C01804=1030.164,-32.787,-88.307,167.818,43.138,158.004
C01805=1030.170,-32.537,-88.320,167.821,43.137,158.004
C01806=1030.176,-32.288,-88.333,167.824,43.135,158.004
C01807=1030.183,-32.038,-88.346,167.827,43.134,158.004
C01808=1030.190,-31.789,-88.359,167.829,43.132,158.004
C01809=1030.196,-31.539,-88.372,167.832,43.130,158.004
C01810=1030.202,-31.290,-88.385,167.834,43.129,158.004
C01811=1030.208,-31.040,-88.398,167.836,43.128,158.004
C01812=1030.214,-30.790,-88.411,167.839,43.126,158.004
C01813=1030.221,-30.540,-88.424,167.842,43.125,158.004
C01814=1030.227,-30.291,-88.438,167.845,43.123,158.004
C01815=1030.233,-30.042,-88.451,167.847,43.122,158.004
C01816=1030.239,-29.792,-88.464,167.850,43.120,158.004
C01817=1030.245,-29.543,-88.477,167.853,43.119,158.003
C01818=1030.252,-29.293,-88.490,167.856,43.117,158.003
C01819=1030.258,-29.044,-88.504,167.858,43.116,158.003
C01820=1030.264,-28.794,-88.516,167.860,43.114,158.003
C01821=1030.270,-28.544,-88.530,167.863,43.113,158.003
C01822=1030.277,-28.294,-88.544,167.866,43.111,158.003
C01823=1030.283,-28.045,-88.557,167.868,43.110,158.003
C01824=1030.289,-27.795,-88.570,167.871,43.108,158.003
C01825=1030.295,-27.546,-88.583,167.874,43.107,158.003
C01826=1030.302,-27.296,-88.596,167.877,43.105,158.003
C01827=1030.308,-27.046,-88.610,167.879,43.104,158.003
C01828=1030.314,-26.797,-88.623,167.881,43.102,158.003
C01829=1030.320,-26.548,-88.636,167.884,43.101,158.003
C01830=1030.326,-26.298,-88.651,167.887,43.099,158.002
C01831=1030.333,-26.048,-88.664,167.889,43.098,158.002
C01832=1030.339,-25.798,-88.676,167.892,43.097,158.002
C01833=1030.345,-25.549,-88.690,167.895,43.095,158.002
C01834=1030.351,-25.299,-88.704,167.897,43.094,158.002
C01835=1030.357,-25.050,-88.717,167.899,43.092,158.002
C01836=1030.363,-24.800,-88.730,167.902,43.091,158.002
C01837=1030.369,-24.551,-88.744,167.905,43.090,158.002
C01838=1030.376,-24.301,-88.758,167.908,43.088,158.002
C01839=1030.382,-24.052,-88.771,167.911,43.087,158.002
C01840=1030.388,-23.802,-88.784,167.912,43.085,158.002
C01841=1030.394,-23.552,-88.799,167.915,43.084,158.002
C01842=1030.400,-23.303,-88.812,167.918,43.083,158.002
C01843=1030.406,-23.054,-88.825,167.921,43.081,158.002
C01844=1030.413,-22.804,-88.838,167.923,43.080,158.002
C01845=1030.419,-22.554,-88.853,167.925,43.078,158.002
C01846=1030.425,-22.305,-88.866,167.928,43.077,158.002
C01847=1030.431,-22.055,-88.879,167.931,43.075,158.001
C01848=1030.437,-21.805,-88.893,167.933,43.074,158.002
C01849=1030.443,-21.556,-88.907,167.936,43.072,158.001
C01850=1030.450,-21.307,-88.921,167.939,43.071,158.001
C01851=1030.457,-21.057,-88.934,167.941,43.070,158.001
C01852=1030.462,-20.808,-88.948,167.943,43.068,158.001
C01853=1030.469,-20.526,-88.963,167.946,43.067,158.001
C01854=1030.477,-20.245,-88.978,167.950,43.065,158.001
C01855=1030.484,-19.963,-88.994,167.953,43.063,158.001
C01856=1030.491,-19.682,-89.010,167.956,43.062,158.001
C01857=1030.497,-19.432,-89.023,167.958,43.060,158.001
C01858=1030.503,-19.182,-89.037,167.961,43.059,158.001
C01859=1030.510,-18.934,-89.051,167.963,43.057,158.001
C01860=1030.516,-18.684,-89.064,167.965,43.056,158.001
C01861=1030.522,-18.434,-89.079,167.968,43.054,158.001
C01862=1030.528,-18.185,-89.092,167.971,43.053,158.001
C01863=1030.535,-17.935,-89.105,167.974,43.051,158.000
C01864=1030.541,-17.685,-89.119,167.977,43.050,158.000
C01865=1030.547,-17.437,-89.133,167.978,43.048,158.000
C01866=1030.554,-17.187,-89.147,167.981,43.047,158.000
C01867=1030.560,-16.937,-89.160,167.984,43.045,158.000
C01868=1030.566,-16.687,-89.174,167.986,43.044,158.000
C01869=1030.572,-16.438,-89.188,167.989,43.042,158.000
C01870=1030.579,-16.188,-89.202,167.991,43.041,158.000
C01871=1030.585,-15.939,-89.216,167.994,43.039,158.000
C01872=1030.592,-15.689,-89.230,167.996,43.038,158.000
C01873=1030.598,-15.440,-89.243,167.999,43.037,158.000
C01874=1030.604,-15.190,-89.258,168.002,43.035,158.000
C01875=1030.610,-14.940,-89.272,168.004,43.034,158.000
C01876=1030.616,-14.691,-89.285,168.007,43.033,158.000
C01877=1030.622,-14.441,-89.300,168.009,43.031,158.000
C01878=1030.628,-14.192,-89.313,168.012,43.030,158.000
C01879=1030.635,-13.942,-89.327,168.014,43.029,158.000
C01880=1030.641,-13.693,-89.341,168.017,43.027,157.999
C01881=1030.647,-13.443,-89.356,168.020,43.026,157.999
C01882=1030.653,-13.194,-89.370,168.022,43.025,157.999
C01883=1030.660,-12.944,-89.384,168.024,43.023,157.999
C01884=1030.665,-12.694,-89.398,168.027,43.022,157.999
C01885=1030.672,-12.445,-89.412,168.030,43.021,157.999
C01886=1030.678,-12.196,-89.426,168.032,43.019,157.999
C01887=1030.684,-11.946,-89.441,168.034,43.018,157.999
C01888=1030.690,-11.697,-89.454,168.037,43.016,157.999
C01889=1030.697,-11.447,-89.469,168.040,43.015,157.999
C01890=1030.703,-11.198,-89.482,168.043,43.014,157.999
C01891=1030.709,-10.947,-89.496,168.044,43.012,157.999
C01892=1030.716,-10.699,-89.510,168.047,43.011,157.999
C01893=1030.722,-10.449,-89.525,168.050,43.010,157.999
C01894=1030.727,-10.200,-89.539,168.053,43.008,157.999
C01895=1030.734,-9.950,-89.553,168.054,43.007,157.999
C01896=1030.740,-9.701,-89.567,168.057,43.005,157.998
C01897=1030.747,-9.451,-89.581,168.060,43.004,157.998
C01898=1030.753,-9.202,-89.596,168.063,43.003,157.998
C01899=1030.759,-8.951,-89.610,168.064,43.001,157.998
C01900=1030.766,-8.702,-89.624,168.067,43.000,157.998
C01901=1030.771,-8.453,-89.638,168.070,42.999,157.998
C01902=1030.778,-8.203,-89.653,168.073,42.997,157.998
C01903=1030.784,-7.954,-89.667,168.075,42.996,157.998
C01904=1030.790,-7.704,-89.681,168.077,42.994,157.998
C01905=1030.797,-7.455,-89.695,168.080,42.993,157.998
C01906=1030.803,-7.205,-89.710,168.083,42.992,157.998
C01907=1030.810,-6.956,-89.724,168.085,42.990,157.998
C01908=1030.816,-6.706,-89.738,168.087,42.989,157.998
C01909=1030.822,-6.456,-89.753,168.090,42.987,157.998
C01910=1030.829,-6.207,-89.767,168.092,42.986,157.998
C01911=1030.835,-5.958,-89.781,168.095,42.985,157.998
C01912=1030.841,-5.708,-89.796,168.097,42.983,157.997
C01913=1030.847,-5.459,-89.810,168.100,42.982,157.997
C01914=1030.853,-5.209,-89.824,168.102,42.980,157.997
C01915=1030.861,-4.960,-89.838,168.105,42.979,157.997
C01916=1030.866,-4.710,-89.852,168.107,42.977,157.997
C01917=1030.873,-4.427,-89.869,168.110,42.976,157.997
C01918=1030.881,-4.144,-89.885,168.113,42.974,157.997
C01919=1030.888,-3.861,-89.901,168.116,42.973,157.997
C01920=1030.895,-3.578,-89.918,168.118,42.971,157.997
C01921=1030.901,-3.328,-89.932,168.121,42.970,157.997
C01922=1030.907,-3.079,-89.947,168.124,42.969,157.997
C01923=1030.913,-2.830,-89.962,168.126,42.968,157.997
C01924=1030.920,-2.580,-89.977,168.129,42.966,157.997
C01925=1030.926,-2.331,-89.991,168.131,42.965,157.997
C01926=1030.932,-2.081,-90.006,168.133,42.964,157.997
C01927=1030.938,-1.831,-90.021,168.136,42.963,157.997
C01928=1030.944,-1.582,-90.035,168.139,42.961,157.997
C01929=1030.950,-1.332,-90.050,168.141,42.960,157.997
C01930=1030.957,-1.083,-90.065,168.144,42.959,157.997
C01931=1030.962,-0.834,-90.080,168.146,42.958,157.997
C01932=1030.969,-0.584,-90.095,168.148,42.956,157.996
C01933=1030.975,-0.334,-90.110,168.151,42.955,157.996
C01934=1030.981,-0.085,-90.123,168.154,42.954,157.996
C01935=1030.987,0.165,-90.138,168.156,42.953,157.996
C01936=1030.993,0.414,-90.153,168.158,42.951,157.996
C01937=1030.999,0.663,-90.168,168.160,42.950,157.996
C01938=1031.006,0.913,-90.183,168.163,42.949,157.996
C01939=1031.013,1.162,-90.197,168.166,42.948,157.996
C01940=1031.018,1.411,-90.212,168.167,42.946,157.996
C01941=1031.025,1.661,-90.227,168.170,42.945,157.996
C01942=1031.031,1.911,-90.242,168.173,42.944,157.996
C01943=1031.038,2.160,-90.257,168.175,42.943,157.996
C01944=1031.043,2.409,-90.271,168.178,42.941,157.996
C01945=1031.050,2.659,-90.286,168.180,42.940,157.996
C01946=1031.056,2.909,-90.301,168.182,42.939,157.996
C01947=1031.063,3.158,-90.316,168.185,42.938,157.996
C01948=1031.068,3.407,-90.331,168.188,42.936,157.996
C01949=1031.075,3.657,-90.346,168.190,42.935,157.996
C01950=1031.081,3.907,-90.361,168.192,42.934,157.996
C01951=1031.087,4.156,-90.375,168.195,42.932,157.995
C01952=1031.093,4.405,-90.390,168.197,42.931,157.995
C01953=1031.100,4.655,-90.405,168.200,42.930,157.995
C01954=1031.106,4.904,-90.420,168.203,42.929,157.995
C01955=1031.112,5.154,-90.435,168.204,42.927,157.995
C01956=1031.118,5.403,-90.449,168.207,42.926,157.995
C01957=1031.125,5.653,-90.464,168.210,42.925,157.995
C01958=1031.131,5.902,-90.479,168.212,42.923,157.995
C01959=1031.137,6.152,-90.494,168.214,42.922,157.995
C01960=1031.144,6.402,-90.509,168.217,42.921,157.995
C01961=1031.149,6.651,-90.524,168.219,42.919,157.995
C01962=1031.156,6.900,-90.539,168.222,42.918,157.995
C01963=1031.162,7.150,-90.554,168.225,42.917,157.995
C01964=1031.169,7.400,-90.569,168.226,42.915,157.995
C01965=1031.175,7.649,-90.584,168.229,42.914,157.995
C01966=1031.182,7.898,-90.599,168.231,42.913,157.995
C01967=1031.187,8.147,-90.614,168.234,42.911,157.994
C01968=1031.194,8.397,-90.629,168.237,42.910,157.994
C01969=1031.200,8.647,-90.644,168.238,42.909,157.994
C01970=1031.207,8.896,-90.659,168.241,42.907,157.994
C01971=1031.213,9.146,-90.674,168.244,42.906,157.994
C01972=1031.220,9.395,-90.689,168.246,42.905,157.994
C01973=1031.226,9.645,-90.704,168.248,42.903,157.994
C01974=1031.232,9.894,-90.719,168.251,42.902,157.994
C01975=1031.238,10.143,-90.734,168.253,42.901,157.994
C01976=1031.245,10.393,-90.749,168.256,42.899,157.994
C01977=1031.251,10.642,-90.764,168.259,42.898,157.994
C01978=1031.257,10.892,-90.780,168.260,42.897,157.994
C01979=1031.263,11.142,-90.795,168.263,42.895,157.994
C01980=1031.270,11.391,-90.810,168.266,42.894,157.994
C01981=1031.277,11.675,-90.827,168.269,42.892,157.994
C01982=1031.285,11.961,-90.844,168.271,42.891,157.994
C01983=1031.292,12.245,-90.862,168.274,42.889,157.993
C01984=1031.299,12.531,-90.878,168.277,42.888,157.993
C01985=1031.306,12.780,-90.894,168.279,42.886,157.993
C01986=1031.312,13.030,-90.909,168.281,42.885,157.993
C01987=1031.319,13.279,-90.924,168.284,42.883,157.993
C01988=1031.325,13.529,-90.939,168.286,42.882,157.993
C01989=1031.332,13.778,-90.955,168.289,42.881,157.993
C01990=1031.338,14.028,-90.970,168.291,42.879,157.993
C01991=1031.344,14.278,-90.985,168.293,42.878,157.993
C01992=1031.350,14.527,-91.001,168.296,42.877,157.993
C01993=1031.357,14.776,-91.016,168.298,42.876,157.993
C01994=1031.362,15.025,-91.032,168.301,42.875,157.993
C01995=1031.368,15.275,-91.047,168.303,42.873,157.993
C01996=1031.375,15.524,-91.062,168.305,42.872,157.993
C01997=1031.381,15.774,-91.078,168.308,42.871,157.993
C01998=1031.387,16.023,-91.093,168.310,42.870,157.993
C01999=1031.394,16.272,-91.108,168.313,42.868,157.992
C02000=1031.400,16.522,-91.123,168.315,42.867,157.992
C02001=1031.406,16.771,-91.140,168.317,42.866,157.992
C02002=1031.413,17.021,-91.155,168.320,42.865,157.992
C02003=1031.419,17.270,-91.170,168.322,42.863,157.992
C02004=1031.425,17.520,-91.186,168.325,42.862,157.992
C02005=1031.432,17.769,-91.201,168.326,42.861,157.992
C02006=1031.438,18.019,-91.216,168.329,42.860,157.992
C02007=1031.444,18.268,-91.233,168.332,42.858,157.992
C02008=1031.450,18.518,-91.248,168.334,42.857,157.992
C02009=1031.457,18.767,-91.263,168.337,42.856,157.992
C02010=1031.463,19.017,-91.279,168.338,42.855,157.992
C02011=1031.469,19.266,-91.294,168.341,42.853,157.992
C02012=1031.476,19.515,-91.309,168.344,42.852,157.992
C02013=1031.482,19.765,-91.326,168.346,42.851,157.992
C02014=1031.488,20.014,-91.341,168.348,42.849,157.992
C02015=1031.494,20.264,-91.357,168.350,42.848,157.991
C02016=1031.500,20.513,-91.372,168.353,42.847,157.991
C02017=1031.507,20.762,-91.387,168.355,42.846,157.991
C02018=1031.513,21.012,-91.404,168.358,42.845,157.991
C02019=1031.519,21.261,-91.419,168.361,42.843,157.991
C02020=1031.525,21.511,-91.435,168.362,42.842,157.991
C02021=1031.532,21.760,-91.451,168.365,42.841,157.991
C02022=1031.538,22.010,-91.466,168.367,42.840,157.991
C02023=1031.544,22.259,-91.482,168.370,42.839,157.991
C02024=1031.550,22.508,-91.498,168.372,42.837,157.991
C02025=1031.557,22.759,-91.513,168.374,42.836,157.991
C02026=1031.563,23.008,-91.530,168.376,42.835,157.991
C02027=1031.570,23.257,-91.545,168.379,42.834,157.991
C02028=1031.576,23.507,-91.560,168.382,42.832,157.991
C02029=1031.582,23.756,-91.576,168.384,42.831,157.991
C02030=1031.589,24.005,-91.592,168.386,42.830,157.991
C02031=1031.595,24.255,-91.608,168.388,42.829,157.991
C02032=1031.601,24.504,-91.623,168.391,42.827,157.991
C02033=1031.607,24.753,-91.640,168.393,42.826,157.991
C02034=1031.614,25.002,-91.655,168.396,42.825,157.991
C02035=1031.620,25.252,-91.671,168.398,42.824,157.991
C02036=1031.626,25.501,-91.686,168.400,42.822,157.990
C02037=1031.633,25.751,-91.703,168.403,42.821,157.990
C02038=1031.640,26.000,-91.719,168.405,42.820,157.990
C02039=1031.645,26.250,-91.734,168.408,42.819,157.990
C02040=1031.652,26.499,-91.750,168.409,42.817,157.990
C02041=1031.658,26.749,-91.766,168.412,42.816,157.990
C02042=1031.665,26.998,-91.782,168.414,42.815,157.990
C02043=1031.670,27.247,-91.798,168.417,42.814,157.990
C02044=1031.677,27.497,-91.813,168.419,42.812,157.990
C02045=1031.684,27.783,-91.832,168.421,42.811,157.990
C02046=1031.692,28.069,-91.850,168.424,42.810,157.990
C02047=1031.699,28.356,-91.869,168.427,42.808,157.990
C02048=1031.706,28.642,-91.887,168.430,42.807,157.990
C02049=1031.712,28.892,-91.903,168.432,42.806,157.990
C02050=1031.718,29.141,-91.919,168.434,42.805,157.990
C02051=1031.725,29.390,-91.935,168.437,42.803,157.989
C02052=1031.731,29.640,-91.951,168.439,42.802,157.989
C02053=1031.737,29.889,-91.968,168.442,42.801,157.989
C02054=1031.743,30.138,-91.984,168.444,42.800,157.989
C02055=1031.750,30.388,-92.000,168.446,42.799,157.989
C02056=1031.756,30.637,-92.016,168.448,42.798,157.989
C02057=1031.762,30.887,-92.032,168.451,42.796,157.989
C02058=1031.768,31.136,-92.048,168.453,42.795,157.989
C02059=1031.774,31.385,-92.064,168.456,42.794,157.989
C02060=1031.780,31.634,-92.081,168.457,42.793,157.989
C02061=1031.787,31.884,-92.097,168.460,42.792,157.989
C02062=1031.794,32.133,-92.113,168.462,42.790,157.989
C02063=1031.800,32.383,-92.129,168.465,42.789,157.989
C02064=1031.806,32.632,-92.145,168.468,42.788,157.989
C02065=1031.812,32.881,-92.161,168.469,42.787,157.989
C02066=1031.819,33.131,-92.178,168.472,42.786,157.989
C02067=1031.825,33.381,-92.194,168.474,42.784,157.989
C02068=1031.831,33.630,-92.210,168.477,42.783,157.989
C02069=1031.837,33.879,-92.226,168.479,42.782,157.989
C02070=1031.843,34.128,-92.242,168.481,42.781,157.989
C02071=1031.850,34.378,-92.259,168.483,42.780,157.989
C02072=1031.856,34.628,-92.275,168.486,42.778,157.988
C02073=1031.862,34.877,-92.291,168.488,42.777,157.988
C02074=1031.868,35.126,-92.307,168.491,42.776,157.988
C02075=1031.875,35.376,-92.323,168.492,42.775,157.988
C02076=1031.882,35.625,-92.340,168.495,42.774,157.988
C02077=1031.888,35.874,-92.356,168.497,42.772,157.988
C02078=1031.894,36.123,-92.372,168.500,42.771,157.988
C02079=1031.900,36.373,-92.389,168.502,42.770,157.988
C02080=1031.907,36.622,-92.405,168.504,42.769,157.988
C02081=1031.913,36.872,-92.421,168.506,42.767,157.988
C02082=1031.920,37.122,-92.438,168.509,42.766,157.988
C02083=1031.926,37.371,-92.454,168.511,42.765,157.988
C02084=1031.932,37.620,-92.471,168.514,42.764,157.988
C02085=1031.938,37.869,-92.487,168.515,42.763,157.988
C02086=1031.944,38.119,-92.504,168.518,42.762,157.988
C02087=1031.950,38.369,-92.520,168.520,42.760,157.988
C02088=1031.957,38.617,-92.537,168.523,42.759,157.988
C02089=1031.963,38.867,-92.553,168.525,42.758,157.987
C02090=1031.969,39.117,-92.570,168.528,42.757,157.987
C02091=1031.975,39.366,-92.586,168.529,42.756,157.987
C02092=1031.981,39.615,-92.603,168.532,42.755,157.987
C02093=1031.988,39.865,-92.620,168.534,42.754,157.987
C02094=1031.994,40.114,-92.636,168.537,42.753,157.987
C02095=1032.001,40.363,-92.652,168.539,42.751,157.987
C02096=1032.007,40.613,-92.669,168.541,42.750,157.987
C02097=1032.013,40.862,-92.685,168.543,42.749,157.987
C02098=1032.019,41.111,-92.701,168.546,42.748,157.987
C02099=1032.026,41.361,-92.719,168.548,42.747,157.987
C02100=1032.032,41.610,-92.735,168.551,42.746,157.987
C02101=1032.038,41.859,-92.751,168.553,42.745,157.987
C02102=1032.045,42.109,-92.769,168.555,42.743,157.987
C02103=1032.051,42.358,-92.785,168.557,42.742,157.987
C02104=1032.057,42.607,-92.802,168.560,42.741,157.987
C02105=1032.064,42.857,-92.818,168.562,42.740,157.987
C02106=1032.070,43.106,-92.835,168.565,42.739,157.987
C02107=1032.075,43.355,-92.852,168.566,42.738,157.987
C02108=1032.082,43.605,-92.869,168.568,42.737,157.987
C02109=1032.089,43.891,-92.889,168.571,42.736,157.987
C02110=1032.096,44.178,-92.907,168.574,42.734,157.986
C02111=1032.103,44.464,-92.927,168.577,42.733,157.986
C02112=1032.110,44.750,-92.947,168.580,42.732,157.986
C02113=1032.116,45.000,-92.963,168.581,42.731,157.986
C02114=1032.122,45.248,-92.980,168.584,42.730,157.986
C02115=1032.128,45.498,-92.996,168.586,42.729,157.986
C02116=1032.134,45.747,-93.014,168.588,42.728,157.986
C02117=1032.140,45.996,-93.031,168.591,42.726,157.986
C02118=1032.147,46.246,-93.048,168.593,42.725,157.986
C02119=1032.153,46.495,-93.065,168.595,42.724,157.986
C02120=1032.159,46.745,-93.082,168.597,42.723,157.986
C02121=1032.165,46.994,-93.099,168.600,42.722,157.986
C02122=1032.171,47.243,-93.115,168.602,42.721,157.986
C02123=1032.178,47.493,-93.132,168.605,42.720,157.986
C02124=1032.183,47.742,-93.149,168.607,42.719,157.986
C02125=1032.189,47.991,-93.166,168.608,42.717,157.986
C02126=1032.196,48.241,-93.184,168.611,42.716,157.986
C02127=1032.202,48.490,-93.200,168.613,42.715,157.986
C02128=1032.208,48.740,-93.218,168.616,42.714,157.986
C02129=1032.214,48.989,-93.234,168.618,42.713,157.986
C02130=1032.221,49.238,-93.251,168.620,42.712,157.986
C02131=1032.227,49.487,-93.269,168.622,42.711,157.986
C02132=1032.232,49.737,-93.285,168.625,42.710,157.986
C02133=1032.239,49.986,-93.303,168.627,42.709,157.986
C02134=1032.246,50.235,-93.319,168.629,42.708,157.986
C02135=1032.251,50.485,-93.337,168.632,42.707,157.986
C02136=1032.258,50.734,-93.354,168.634,42.706,157.985
C02137=1032.265,50.983,-93.371,168.636,42.705,157.985
C02138=1032.270,51.233,-93.387,168.638,42.703,157.985
C02139=1032.277,51.483,-93.405,168.641,42.702,157.985
C02140=1032.283,51.731,-93.422,168.643,42.701,157.985
C02141=1032.289,51.981,-93.438,168.646,42.700,157.985
C02142=1032.295,52.230,-93.456,168.647,42.699,157.985
C02143=1032.301,52.479,-93.473,168.650,42.698,157.985
C02144=1032.308,52.729,-93.491,168.652,42.697,157.985
C02145=1032.314,52.978,-93.507,168.654,42.696,157.985
C02146=1032.320,53.228,-93.525,168.657,42.695,157.985
C02147=1032.326,53.476,-93.542,168.658,42.693,157.985
C02148=1032.333,53.726,-93.558,168.661,42.692,157.985
C02149=1032.338,53.975,-93.576,168.663,42.691,157.985
C02150=1032.345,54.225,-93.593,168.666,42.690,157.985
C02151=1032.352,54.474,-93.610,168.668,42.689,157.985
C02152=1032.358,54.723,-93.628,168.671,42.688,157.985
C02153=1032.364,54.973,-93.645,168.672,42.687,157.985
C02154=1032.370,55.222,-93.662,168.675,42.685,157.985
C02155=1032.377,55.472,-93.679,168.677,42.684,157.984
C02156=1032.383,55.721,-93.697,168.680,42.683,157.984
C02157=1032.390,55.970,-93.714,168.682,42.682,157.984
C02158=1032.396,56.219,-93.730,168.684,42.681,157.984
C02159=1032.402,56.469,-93.748,168.686,42.680,157.984
C02160=1032.408,56.718,-93.765,168.688,42.678,157.984
C02161=1032.415,56.967,-93.783,168.691,42.677,157.984
C02162=1032.421,57.216,-93.800,168.693,42.676,157.984
C02163=1032.427,57.466,-93.818,168.696,42.675,157.984
C02164=1032.434,57.716,-93.834,168.697,42.674,157.984
C02165=1032.440,57.965,-93.851,168.700,42.673,157.984
C02166=1032.446,58.214,-93.869,168.702,42.671,157.984
C02167=1032.452,58.463,-93.886,168.705,42.670,157.984
C02168=1032.459,58.712,-93.903,168.707,42.669,157.984
C02169=1032.465,58.962,-93.921,168.709,42.668,157.984
C02170=1032.472,59.211,-93.938,168.711,42.667,157.984
C02171=1032.479,59.460,-93.956,168.714,42.666,157.984
C02172=1032.484,59.710,-93.972,168.716,42.664,157.983
C02173=1032.492,59.996,-93.993,168.719,42.663,157.983
C02174=1032.499,60.282,-94.013,168.721,42.662,157.983
C02175=1032.506,60.568,-94.033,168.724,42.660,157.983
C02176=1032.514,60.853,-94.052,168.726,42.659,157.983
C02177=1032.520,61.103,-94.070,168.729,42.658,157.983
C02178=1032.526,61.352,-94.087,168.730,42.656,157.983
C02179=1032.533,61.601,-94.104,168.733,42.655,157.983
C02180=1032.539,61.851,-94.122,168.735,42.654,157.983
C02181=1032.546,62.100,-94.139,168.738,42.653,157.983
C02182=1032.552,62.349,-94.157,168.740,42.651,157.983
C02183=1032.559,62.599,-94.175,168.742,42.650,157.983
C02184=1032.565,62.847,-94.192,168.744,42.649,157.983
C02185=1032.572,63.097,-94.209,168.747,42.648,157.983
C02186=1032.578,63.347,-94.227,168.749,42.647,157.983
C02187=1032.584,63.595,-94.244,168.752,42.645,157.982
C02188=1032.590,63.845,-94.262,168.753,42.644,157.982
C02189=1032.597,64.094,-94.279,168.756,42.643,157.982
C02190=1032.603,64.344,-94.297,168.758,42.642,157.982
C02191=1032.609,64.593,-94.315,168.761,42.641,157.982
C02192=1032.616,64.843,-94.332,168.763,42.640,157.982
C02193=1032.621,65.092,-94.349,168.765,42.639,157.982
C02194=1032.628,65.341,-94.368,168.768,42.638,157.982
C02195=1032.634,65.590,-94.385,168.769,42.637,157.982
C02196=1032.640,65.839,-94.403,168.772,42.636,157.982
C02197=1032.647,66.089,-94.420,168.774,42.635,157.982
C02198=1032.653,66.339,-94.438,168.777,42.633,157.982
C02199=1032.659,66.587,-94.455,168.779,42.632,157.982
C02200=1032.666,66.836,-94.474,168.780,42.631,157.982
C02201=1032.672,67.086,-94.492,168.783,42.630,157.982
C02202=1032.678,67.335,-94.509,168.785,42.629,157.982
C02203=1032.684,67.585,-94.527,168.788,42.628,157.982
C02204=1032.690,67.834,-94.545,168.790,42.627,157.982
C02205=1032.697,68.083,-94.563,168.793,42.626,157.982
C02206=1032.703,68.332,-94.580,168.794,42.625,157.982
C02207=1032.709,68.582,-94.598,168.797,42.624,157.982
C02208=1032.715,68.831,-94.617,168.799,42.623,157.982
C02209=1032.722,69.080,-94.634,168.801,42.622,157.982
C02210=1032.728,69.329,-94.652,168.804,42.621,157.982
C02211=1032.734,69.579,-94.670,168.805,42.619,157.981
C02212=1032.740,69.828,-94.688,168.808,42.618,157.981
C02213=1032.747,70.077,-94.705,168.810,42.617,157.981
C02214=1032.753,70.327,-94.723,168.813,42.616,157.981
C02215=1032.759,70.576,-94.742,168.815,42.615,157.981
C02216=1032.765,70.826,-94.760,168.817,42.614,157.981
C02217=1032.771,71.075,-94.777,168.820,42.613,157.981
C02218=1032.778,71.324,-94.795,168.821,42.612,157.981
C02219=1032.784,71.573,-94.813,168.824,42.611,157.981
C02220=1032.790,71.822,-94.832,168.826,42.610,157.981
C02221=1032.796,72.071,-94.850,168.828,42.609,157.981
C02222=1032.802,72.321,-94.868,168.831,42.608,157.981
C02223=1032.809,72.570,-94.886,168.833,42.607,157.981
C02224=1032.815,72.820,-94.904,168.835,42.606,157.981
C02225=1032.821,73.047,-94.920,168.837,42.605,157.981
C02226=1032.826,73.274,-94.937,168.839,42.604,157.981
C02227=1032.832,73.502,-94.954,168.841,42.603,157.981
C02228=1032.838,73.729,-94.970,168.844,42.602,157.981
C02229=1032.843,73.957,-94.986,168.846,42.601,157.981
C02230=1032.849,74.185,-95.003,168.847,42.600,157.981
C02231=1032.854,74.412,-95.020,168.849,42.599,157.981
C02232=1032.860,74.639,-95.036,168.851,42.598,157.980
C02233=1032.866,74.889,-95.054,168.854,42.597,157.980
C02234=1032.873,75.138,-95.072,168.856,42.596,157.980
C02235=1032.879,75.387,-95.090,168.859,42.594,157.980
C02236=1032.886,75.636,-95.108,168.860,42.593,157.980
C02237=1032.893,75.966,-95.133,168.863,42.592,157.980
C02238=1032.902,76.295,-95.157,168.867,42.590,157.980
C02239=1032.910,76.624,-95.180,168.870,42.589,157.980
C02240=1032.918,76.953,-95.204,168.873,42.587,157.980
C02241=1032.925,77.202,-95.223,168.875,42.586,157.980
C02242=1032.931,77.452,-95.241,168.877,42.585,157.980
C02243=1032.937,77.701,-95.259,168.879,42.584,157.980
C02244=1032.943,77.950,-95.278,168.882,42.583,157.980
C02245=1032.949,78.200,-95.296,168.884,42.582,157.980
C02246=1032.956,78.449,-95.314,168.887,42.581,157.980
C02247=1032.962,78.698,-95.332,168.889,42.581,157.980
C02248=1032.968,78.947,-95.351,168.890,42.580,157.980
C02249=1032.975,79.197,-95.370,168.893,42.579,157.980
C02250=1032.980,79.447,-95.388,168.895,42.578,157.980
C02251=1032.986,79.695,-95.406,168.898,42.577,157.980
C02252=1032.992,79.944,-95.425,168.900,42.576,157.980
C02253=1032.998,80.194,-95.443,168.902,42.575,157.980
C02254=1033.005,80.443,-95.462,168.905,42.574,157.980
C02255=1033.011,80.692,-95.480,168.906,42.573,157.980
C02256=1033.018,80.941,-95.499,168.909,42.571,157.980
C02257=1033.023,81.190,-95.516,168.911,42.571,157.980
C02258=1033.029,81.440,-95.536,168.913,42.570,157.979
C02259=1033.035,81.689,-95.554,168.916,42.568,157.979
C02260=1033.042,81.938,-95.573,168.918,42.567,157.979
C02261=1033.048,82.188,-95.591,168.920,42.566,157.979
C02262=1033.054,82.437,-95.610,168.922,42.565,157.979
C02263=1033.061,82.686,-95.628,168.925,42.564,157.979
C02264=1033.067,82.935,-95.647,168.927,42.563,157.979
C02265=1033.072,83.185,-95.665,168.929,42.562,157.979
C02266=1033.078,83.434,-95.684,168.932,42.561,157.979
C02267=1033.085,83.683,-95.702,168.933,42.560,157.979
C02268=1033.091,83.932,-95.721,168.936,42.559,157.979
C02269=1033.098,84.181,-95.740,168.938,42.558,157.979
C02270=1033.104,84.431,-95.758,168.941,42.557,157.979
C02271=1033.110,84.680,-95.776,168.943,42.556,157.979
C02272=1033.116,84.929,-95.795,168.945,42.555,157.979
C02273=1033.122,85.178,-95.814,168.948,42.554,157.979
C02274=1033.129,85.428,-95.833,168.949,42.553,157.979
C02275=1033.135,85.677,-95.851,168.952,42.552,157.979
C02276=1033.141,85.926,-95.869,168.954,42.551,157.979
C02277=1033.148,86.176,-95.888,168.957,42.550,157.979
C02278=1033.153,86.425,-95.907,168.959,42.549,157.979
C02279=1033.160,86.674,-95.926,168.961,42.548,157.979
C02280=1033.166,86.923,-95.945,168.963,42.547,157.979
C02281=1033.173,87.172,-95.963,168.965,42.546,157.979
C02282=1033.179,87.421,-95.982,168.968,42.545,157.979
C02283=1033.185,87.671,-96.000,168.970,42.544,157.978
C02284=1033.191,87.920,-96.020,168.973,42.543,157.978
C02285=1033.197,88.170,-96.038,168.975,42.542,157.978
C02286=1033.204,88.419,-96.056,168.977,42.540,157.978
C02287=1033.210,88.668,-96.075,168.979,42.539,157.978
C02288=1033.217,88.917,-96.094,168.981,42.538,157.978
C02289=1033.223,89.166,-96.112,168.984,42.537,157.978
C02290=1033.229,89.416,-96.131,168.986,42.536,157.978
C02291=1033.235,89.665,-96.150,168.989,42.535,157.978
C02292=1033.241,89.914,-96.169,168.990,42.534,157.978
C02293=1033.248,90.163,-96.187,168.993,42.533,157.978
C02294=1033.254,90.412,-96.207,168.995,42.532,157.978
C02295=1033.260,90.662,-96.225,168.997,42.531,157.978
C02296=1033.266,90.911,-96.245,169.000,42.530,157.978
C02297=1033.272,91.160,-96.263,169.002,42.529,157.978
C02298=1033.278,91.409,-96.283,169.005,42.528,157.978
C02299=1033.285,91.658,-96.302,169.006,42.527,157.978
C02300=1033.290,91.907,-96.321,169.009,42.526,157.978
C02301=1033.297,92.193,-96.342,169.011,42.525,157.978
C02302=1033.304,92.479,-96.365,169.014,42.524,157.978
C02303=1033.311,92.764,-96.385,169.017,42.523,157.978
C02304=1033.319,93.050,-96.408,169.020,42.522,157.978
C02305=1033.325,93.299,-96.427,169.022,42.521,157.978
C02306=1033.331,93.548,-96.446,169.023,42.520,157.978
C02307=1033.337,93.798,-96.465,169.026,42.519,157.978
C02308=1033.343,94.046,-96.484,169.028,42.518,157.978
C02309=1033.349,94.296,-96.503,169.031,42.516,157.978
C02310=1033.356,94.545,-96.522,169.033,42.516,157.977
C02311=1033.361,94.794,-96.541,169.036,42.515,157.978
C02312=1033.368,95.043,-96.560,169.038,42.514,157.978
C02313=1033.373,95.293,-96.579,169.039,42.513,157.977
C02314=1033.380,95.541,-96.599,169.042,42.512,157.977
C02315=1033.386,95.791,-96.618,169.044,42.511,157.977
C02316=1033.392,96.040,-96.636,169.047,42.510,157.977
C02317=1033.398,96.289,-96.656,169.049,42.509,157.977
C02318=1033.405,96.539,-96.675,169.052,42.508,157.977
C02319=1033.412,96.788,-96.694,169.053,42.507,157.977
C02320=1033.417,97.037,-96.713,169.056,42.506,157.977
C02321=1033.424,97.286,-96.732,169.058,42.505,157.977
C02322=1033.430,97.535,-96.752,169.060,42.504,157.977
C02323=1033.436,97.784,-96.771,169.063,42.503,157.977
C02324=1033.442,98.034,-96.790,169.065,42.502,157.977
C02325=1033.448,98.283,-96.808,169.068,42.501,157.977
C02326=1033.454,98.532,-96.828,169.069,42.500,157.977
C02327=1033.461,98.781,-96.847,169.072,42.499,157.977
C02328=1033.467,99.031,-96.867,169.074,42.498,157.977
C02329=1033.474,99.279,-96.886,169.077,42.496,157.977
C02330=1033.479,99.529,-96.905,169.079,42.495,157.977
C02331=1033.486,99.778,-96.924,169.082,42.494,157.977
C02332=1033.492,100.027,-96.944,169.083,42.493,157.977
C02333=1033.498,100.276,-96.963,169.085,42.493,157.977
C02334=1033.505,100.526,-96.982,169.088,42.492,157.977
C02335=1033.511,100.775,-97.002,169.090,42.491,157.977
C02336=1033.516,101.024,-97.021,169.093,42.490,157.977
C02337=1033.522,101.273,-97.041,169.095,42.489,157.977
C02338=1033.529,101.522,-97.060,169.098,42.488,157.977
C02339=1033.535,101.771,-97.080,169.100,42.487,157.977
C02340=1033.540,102.020,-97.099,169.102,42.487,157.977
C02341=1033.547,102.270,-97.120,169.104,42.485,157.977
C02342=1033.553,102.519,-97.138,169.106,42.484,157.977
C02343=1033.559,102.768,-97.158,169.109,42.483,157.977
C02344=1033.565,103.017,-97.177,169.111,42.482,157.976
C02345=1033.571,103.266,-97.197,169.114,42.481,157.976
C02346=1033.577,103.515,-97.216,169.116,42.481,157.977
C02347=1033.584,103.765,-97.236,169.118,42.480,157.977
C02348=1033.590,104.014,-97.256,169.121,42.479,157.976
C02349=1033.596,104.263,-97.276,169.122,42.478,157.976
C02350=1033.602,104.512,-97.294,169.125,42.477,157.976
C02351=1033.608,104.761,-97.314,169.127,42.476,157.976
C02352=1033.614,105.011,-97.334,169.130,42.475,157.976
C02353=1033.620,105.260,-97.354,169.132,42.474,157.976
C02354=1033.626,105.509,-97.373,169.135,42.473,157.976
C02355=1033.633,105.758,-97.392,169.137,42.472,157.976
C02356=1033.639,106.007,-97.412,169.138,42.471,157.976
C02357=1033.645,106.257,-97.432,169.141,42.470,157.976
C02358=1033.651,106.505,-97.452,169.143,42.469,157.976
C02359=1033.658,106.755,-97.470,169.146,42.468,157.976
C02360=1033.664,107.003,-97.490,169.148,42.467,157.976
C02361=1033.670,107.253,-97.511,169.151,42.466,157.976
C02362=1033.676,107.502,-97.530,169.153,42.466,157.976
C02363=1033.682,107.751,-97.550,169.156,42.465,157.976
C02364=1033.689,108.000,-97.569,169.157,42.464,157.976
C02365=1033.695,108.286,-97.592,169.160,42.463,157.976
C02366=1033.703,108.571,-97.615,169.163,42.461,157.976
C02367=1033.710,108.857,-97.637,169.166,42.460,157.976
C02368=1033.717,109.143,-97.660,169.169,42.459,157.976
C02369=1033.724,109.392,-97.679,169.171,42.458,157.976
C02370=1033.730,109.640,-97.699,169.173,42.457,157.976
C02371=1033.735,109.890,-97.718,169.175,42.456,157.976
C02372=1033.742,110.139,-97.739,169.177,42.455,157.976
C02373=1033.748,110.388,-97.759,169.180,42.454,157.976
C02374=1033.754,110.638,-97.778,169.182,42.453,157.976
C02375=1033.760,110.887,-97.798,169.185,42.452,157.976
C02376=1033.766,111.136,-97.818,169.187,42.452,157.976
C02377=1033.772,111.385,-97.838,169.190,42.451,157.976
C02378=1033.779,111.634,-97.857,169.191,42.450,157.976
C02379=1033.785,111.883,-97.877,169.194,42.449,157.976
C02380=1033.791,112.132,-97.897,169.196,42.448,157.976
C02381=1033.797,112.381,-97.917,169.199,42.446,157.976
C02382=1033.804,112.631,-97.937,169.201,42.446,157.976
C02383=1033.810,112.879,-97.957,169.204,42.445,157.976
C02384=1033.815,113.129,-97.977,169.206,42.444,157.976
C02385=1033.822,113.378,-97.997,169.208,42.443,157.976
C02386=1033.827,113.627,-98.018,169.211,42.443,157.976
C02387=1033.833,113.876,-98.037,169.212,42.442,157.976
C02388=1033.840,114.126,-98.058,169.215,42.441,157.976
C02389=1033.846,114.375,-98.078,169.217,42.440,157.976
C02390=1033.851,114.624,-98.098,169.220,42.439,157.976
C02391=1033.857,114.872,-98.118,169.222,42.438,157.976
C02392=1033.864,115.122,-98.139,169.225,42.437,157.976
C02393=1033.870,115.371,-98.159,169.227,42.437,157.976
C02394=1033.876,115.620,-98.179,169.229,42.436,157.976
C02395=1033.882,115.869,-98.199,169.231,42.435,157.976
C02396=1033.888,116.118,-98.219,169.234,42.434,157.976
C02397=1033.894,116.367,-98.239,169.236,42.433,157.976
C02398=1033.900,116.617,-98.260,169.238,42.432,157.976
C02399=1033.905,116.866,-98.280,169.241,42.431,157.976
C02400=1033.911,117.115,-98.300,169.243,42.431,157.976
C02401=1033.918,117.364,-98.321,169.246,42.430,157.976
C02402=1033.924,117.613,-98.340,169.248,42.429,157.976
C02403=1033.929,117.862,-98.361,169.251,42.428,157.976
C02404=1033.936,118.112,-98.381,169.253,42.427,157.976
C02405=1033.942,118.360,-98.401,169.255,42.426,157.976
C02406=1033.948,118.610,-98.422,169.257,42.425,157.976
C02407=1033.954,118.859,-98.442,169.259,42.425,157.976
C02408=1033.960,119.107,-98.463,169.262,42.424,157.976
C02409=1033.967,119.357,-98.483,169.264,42.423,157.975
C02410=1033.973,119.605,-98.503,169.267,42.422,157.976
C02411=1033.978,119.855,-98.524,169.269,42.422,157.976
C02412=1033.984,120.104,-98.544,169.272,42.420,157.976
C02413=1033.990,120.353,-98.564,169.274,42.419,157.975
C02414=1033.997,120.602,-98.584,169.277,42.419,157.976
C02415=1034.002,120.852,-98.605,169.278,42.418,157.976
C02416=1034.009,121.100,-98.626,169.281,42.417,157.976
C02417=1034.015,121.349,-98.646,169.283,42.416,157.975
C02418=1034.021,121.598,-98.666,169.286,42.415,157.976
C02419=1034.027,121.848,-98.687,169.288,42.415,157.976
C02420=1034.033,122.097,-98.707,169.291,42.413,157.975
C02421=1034.040,122.346,-98.727,169.293,42.412,157.975
C02422=1034.046,122.594,-98.748,169.296,42.412,157.976
C02423=1034.052,122.844,-98.769,169.298,42.411,157.975
C02424=1034.058,123.093,-98.789,169.300,42.410,157.975
C02425=1034.064,123.343,-98.809,169.302,42.409,157.975
C02426=1034.070,123.591,-98.830,169.305,42.409,157.976
C02427=1034.076,123.840,-98.850,169.307,42.408,157.975
C02428=1034.082,124.089,-98.870,169.310,42.406,157.975
C02429=1034.089,124.375,-98.894,169.313,42.405,157.975
C02430=1034.097,124.660,-98.918,169.316,42.404,157.975
C02431=1034.104,124.946,-98.941,169.319,42.404,157.975
C02432=1034.111,125.231,-98.965,169.321,42.403,157.975
C02433=1034.117,125.480,-98.985,169.323,42.402,157.975
C02434=1034.123,125.729,-99.005,169.326,42.401,157.975
C02435=1034.129,125.978,-99.025,169.328,42.400,157.975
C02436=1034.135,126.227,-99.047,169.331,42.399,157.975
C02437=1034.142,126.477,-99.067,169.333,42.398,157.975
C02438=1034.148,126.726,-99.087,169.336,42.397,157.975
C02439=1034.154,126.975,-99.109,169.338,42.396,157.975
C02440=1034.160,127.224,-99.129,169.341,42.396,157.975
C02441=1034.167,127.473,-99.149,169.343,42.395,157.975
C02442=1034.173,127.721,-99.170,169.345,42.394,157.975
C02443=1034.179,127.971,-99.191,169.347,42.393,157.975
C02444=1034.185,128.220,-99.211,169.350,42.392,157.975
C02445=1034.192,128.469,-99.232,169.353,42.391,157.975
C02446=1034.197,128.718,-99.252,169.355,42.390,157.975
C02447=1034.204,128.967,-99.273,169.358,42.389,157.975
C02448=1034.210,129.216,-99.294,169.360,42.388,157.975
C02449=1034.216,129.465,-99.314,169.363,42.388,157.975
C02450=1034.223,129.714,-99.335,169.365,42.387,157.975
C02451=1034.229,129.963,-99.355,169.367,42.386,157.975
C02452=1034.235,130.212,-99.376,169.370,42.384,157.975
C02453=1034.241,130.462,-99.397,169.372,42.383,157.975
C02454=1034.248,130.710,-99.418,169.375,42.383,157.975
C02455=1034.253,130.960,-99.439,169.377,42.382,157.975
C02456=1034.260,131.208,-99.459,169.380,42.381,157.975
C02457=1034.266,131.458,-99.480,169.382,42.381,157.975
C02458=1034.273,131.707,-99.501,169.385,42.380,157.975
C02459=1034.278,131.956,-99.522,169.387,42.379,157.975
C02460=1034.284,132.205,-99.544,169.390,42.378,157.975
C02461=1034.290,132.454,-99.564,169.391,42.377,157.975
C02462=1034.296,132.703,-99.585,169.394,42.377,157.975
C02463=1034.302,132.952,-99.606,169.396,42.376,157.975
C02464=1034.308,133.201,-99.627,169.399,42.375,157.975
C02465=1034.314,133.451,-99.648,169.402,42.374,157.975
C02466=1034.321,133.699,-99.669,169.404,42.373,157.975
C02467=1034.327,133.949,-99.690,169.407,42.373,157.975
C02468=1034.332,134.197,-99.711,169.409,42.372,157.975
C02469=1034.339,134.447,-99.732,169.412,42.371,157.975
C02470=1034.345,134.696,-99.753,169.414,42.370,157.975
C02471=1034.350,134.944,-99.775,169.417,42.369,157.975
C02472=1034.357,135.194,-99.795,169.418,42.368,157.975
C02473=1034.363,135.443,-99.816,169.422,42.368,157.975
C02474=1034.370,135.691,-99.837,169.424,42.367,157.975
C02475=1034.376,135.940,-99.859,169.426,42.366,157.975
C02476=1034.382,136.190,-99.880,169.429,42.365,157.975
C02477=1034.388,136.438,-99.900,169.431,42.364,157.975
C02478=1034.394,136.688,-99.922,169.434,42.364,157.976
C02479=1034.400,136.937,-99.943,169.436,42.363,157.975
C02480=1034.406,137.186,-99.964,169.439,42.362,157.975
C02481=1034.412,137.435,-99.985,169.442,42.361,157.976
C02482=1034.418,137.684,-100.007,169.444,42.360,157.975
C02483=1034.424,137.933,-100.028,169.447,42.360,157.976
C02484=1034.431,138.182,-100.048,169.449,42.359,157.976
C02485=1034.437,138.431,-100.070,169.451,42.358,157.976
C02486=1034.442,138.680,-100.091,169.454,42.357,157.976
C02487=1034.449,138.929,-100.112,169.456,42.357,157.976
C02488=1034.455,139.178,-100.134,169.459,42.356,157.976
C02489=1034.461,139.427,-100.155,169.461,42.355,157.976
C02490=1034.467,139.676,-100.176,169.464,42.355,157.976
C02491=1034.473,139.925,-100.198,169.466,42.354,157.976
C02492=1034.479,140.174,-100.219,169.469,42.353,157.976
C02493=1034.486,140.459,-100.244,169.472,42.352,157.976
C02494=1034.493,140.745,-100.268,169.475,42.351,157.976
C02495=1034.500,141.030,-100.293,169.478,42.351,157.976
C02496=1034.507,141.315,-100.317,169.481,42.349,157.976
C02497=1034.513,141.564,-100.339,169.483,42.349,157.976
C02498=1034.519,141.813,-100.361,169.486,42.348,157.976
C02499=1034.525,142.062,-100.382,169.489,42.348,157.976
C02500=1034.531,142.311,-100.403,169.490,42.347,157.976
C02501=1034.538,142.560,-100.425,169.493,42.346,157.976
C02502=1034.544,142.809,-100.446,169.495,42.345,157.976
C02503=1034.549,143.058,-100.468,169.498,42.345,157.976
C02504=1034.555,143.307,-100.489,169.501,42.344,157.976
C02505=1034.562,143.556,-100.511,169.503,42.343,157.976
C02506=1034.568,143.805,-100.533,169.506,42.342,157.976
C02507=1034.573,144.054,-100.554,169.508,42.341,157.976
C02508=1034.580,144.303,-100.575,169.511,42.341,157.976
C02509=1034.586,144.552,-100.596,169.514,42.340,157.976
C02510=1034.593,144.801,-100.618,169.516,42.339,157.976
C02511=1034.599,145.050,-100.640,169.519,42.338,157.976
C02512=1034.604,145.299,-100.661,169.521,42.338,157.976
C02513=1034.610,145.548,-100.683,169.524,42.337,157.976
C02514=1034.617,145.797,-100.704,169.527,42.336,157.976
C02515=1034.623,146.046,-100.726,169.528,42.336,157.976
C02516=1034.629,146.296,-100.748,169.531,42.335,157.976
C02517=1034.635,146.544,-100.769,169.534,42.334,157.976
C02518=1034.641,146.793,-100.791,169.536,42.334,157.976
C02519=1034.647,147.042,-100.813,169.539,42.333,157.976
C02520=1034.653,147.291,-100.834,169.542,42.332,157.977
C02521=1034.660,147.540,-100.856,169.544,42.331,157.976
C02522=1034.666,147.790,-100.878,169.547,42.331,157.977
C02523=1034.671,148.038,-100.899,169.549,42.330,157.977
C02524=1034.678,148.287,-100.921,169.552,42.329,157.977
C02525=1034.684,148.536,-100.943,169.555,42.329,157.977
C02526=1034.690,148.785,-100.965,169.557,42.328,157.977
C02527=1034.695,149.035,-100.987,169.560,42.327,157.977
C02528=1034.702,149.283,-101.009,169.563,42.326,157.977
C02529=1034.707,149.532,-101.030,169.565,42.326,157.977
C02530=1034.714,149.781,-101.052,169.568,42.326,157.977
C02531=1034.720,150.029,-101.074,169.570,42.325,157.977
C02532=1034.726,150.279,-101.096,169.573,42.324,157.977
C02533=1034.732,150.528,-101.118,169.576,42.323,157.977
C02534=1034.738,150.777,-101.140,169.578,42.323,157.977
C02535=1034.744,151.026,-101.162,169.581,42.322,157.977
C02536=1034.750,151.274,-101.184,169.583,42.321,157.977
C02537=1034.756,151.524,-101.205,169.585,42.321,157.977
C02538=1034.763,151.772,-101.228,169.588,42.320,157.977
C02539=1034.769,152.021,-101.249,169.591,42.319,157.977
C02540=1034.774,152.270,-101.272,169.593,42.319,157.977
C02541=1034.781,152.520,-101.294,169.596,42.318,157.977
C02542=1034.787,152.769,-101.315,169.599,42.317,157.977
C02543=1034.793,153.017,-101.338,169.601,42.316,157.977
C02544=1034.799,153.267,-101.359,169.604,42.316,157.978
C02545=1034.805,153.515,-101.382,169.607,42.316,157.978
C02546=1034.811,153.764,-101.404,169.609,42.315,157.978
C02547=1034.817,154.013,-101.425,169.612,42.314,157.978
C02548=1034.823,154.262,-101.448,169.615,42.313,157.978
C02549=1034.829,154.511,-101.469,169.617,42.313,157.978
C02550=1034.835,154.760,-101.492,169.620,42.312,157.978
C02551=1034.841,155.009,-101.514,169.623,42.311,157.978
C02552=1034.848,155.258,-101.536,169.625,42.311,157.978
C02553=1034.853,155.507,-101.558,169.628,42.310,157.978
C02554=1034.860,155.756,-101.581,169.631,42.310,157.978
C02555=1034.866,156.005,-101.602,169.633,42.309,157.978
C02556=1034.872,156.254,-101.625,169.636,42.309,157.978
C02557=1034.878,156.538,-101.651,169.639,42.307,157.978
C02558=1034.885,156.823,-101.676,169.642,42.307,157.978
C02559=1034.893,157.109,-101.702,169.645,42.307,157.978
C02560=1034.899,157.394,-101.727,169.648,42.305,157.978
C02561=1034.906,157.642,-101.749,169.651,42.305,157.978
C02562=1034.912,157.891,-101.771,169.654,42.305,157.979
C02563=1034.917,158.140,-101.794,169.655,42.304,157.978
C02564=1034.924,158.389,-101.816,169.659,42.303,157.979
C02565=1034.930,158.638,-101.838,169.662,42.303,157.979
C02566=1034.936,158.887,-101.861,169.664,42.302,157.979
C02567=1034.942,159.136,-101.883,169.666,42.301,157.979
C02568=1034.948,159.385,-101.905,169.669,42.301,157.979
C02569=1034.954,159.634,-101.928,169.673,42.300,157.979
C02570=1034.960,159.883,-101.949,169.674,42.299,157.979
C02571=1034.966,160.132,-101.972,169.677,42.299,157.979
C02572=1034.972,160.381,-101.995,169.680,42.298,157.979
C02573=1034.978,160.629,-102.018,169.682,42.298,157.979
C02574=1034.984,160.878,-102.041,169.686,42.298,157.979
C02575=1034.990,161.127,-102.064,169.689,42.297,157.979
C02576=1034.995,161.377,-102.086,169.691,42.297,157.980
C02577=1035.002,161.625,-102.108,169.694,42.297,157.980
C02578=1035.007,161.874,-102.131,169.696,42.295,157.980
C02579=1035.013,162.123,-102.154,169.698,42.295,157.980
C02580=1035.019,162.372,-102.177,169.702,42.295,157.980
C02581=1035.025,162.620,-102.199,169.705,42.294,157.980
C02582=1035.031,162.869,-102.222,169.708,42.294,157.980
C02583=1035.037,163.118,-102.245,169.710,42.293,157.980
C02584=1035.042,163.368,-102.267,169.713,42.293,157.980
C02585=1035.049,163.616,-102.290,169.716,42.293,157.980
C02586=1035.054,163.865,-102.313,169.718,42.292,157.980
C02587=1035.060,164.114,-102.336,169.721,42.292,157.980
C02588=1035.066,164.363,-102.359,169.724,42.291,157.981
C02589=1035.072,164.612,-102.382,169.726,42.291,157.981
C02590=1035.078,164.860,-102.404,169.729,42.290,157.981
C02591=1035.084,165.109,-102.427,169.732,42.289,157.981
C02592=1035.090,165.358,-102.450,169.735,42.289,157.981
C02593=1035.096,165.608,-102.473,169.737,42.289,157.981
C02594=1035.102,165.856,-102.495,169.740,42.288,157.981
C02595=1035.108,166.105,-102.518,169.743,42.288,157.981
C02596=1035.114,166.354,-102.541,169.745,42.287,157.981
C02597=1035.120,166.603,-102.564,169.748,42.287,157.981
C02598=1035.125,166.852,-102.587,169.751,42.287,157.981
C02599=1035.132,167.101,-102.610,169.754,42.286,157.982
C02600=1035.137,167.350,-102.633,169.756,42.286,157.982
C02601=1035.143,167.598,-102.655,169.759,42.285,157.982
C02602=1035.149,167.847,-102.679,169.762,42.285,157.982
C02603=1035.156,168.096,-102.702,169.765,42.284,157.982
C02604=1035.162,168.345,-102.725,169.767,42.283,157.982
C02605=1035.168,168.594,-102.748,169.770,42.283,157.982
C02606=1035.173,168.843,-102.771,169.773,42.283,157.982
C02607=1035.179,169.092,-102.794,169.776,42.282,157.982
C02608=1035.185,169.340,-102.817,169.779,42.282,157.982
C02609=1035.192,169.590,-102.839,169.781,42.281,157.982
C02610=1035.198,169.839,-102.862,169.784,42.281,157.983
C02611=1035.204,170.087,-102.886,169.787,42.280,157.983
C02612=1035.210,170.336,-102.909,169.790,42.280,157.983
C02613=1035.215,170.585,-102.932,169.792,42.280,157.983
C02614=1035.222,170.833,-102.954,169.795,42.279,157.983
C02615=1035.228,171.083,-102.977,169.798,42.279,157.983
C02616=1035.234,171.331,-103.001,169.801,42.278,157.983
C02617=1035.240,171.580,-103.024,169.804,42.278,157.983
C02618=1035.246,171.829,-103.047,169.806,42.278,157.983
C02619=1035.253,172.078,-103.070,169.810,42.277,157.983
C02620=1035.258,172.327,-103.093,169.812,42.276,157.983
C02621=1035.265,172.611,-103.120,169.815,42.276,157.984
C02622=1035.272,172.895,-103.146,169.818,42.275,157.984
C02623=1035.279,173.180,-103.172,169.823,42.274,157.984
C02624=1035.286,173.464,-103.199,169.826,42.274,157.984
C02625=1035.292,173.713,-103.222,169.829,42.274,157.984
C02626=1035.298,173.963,-103.245,169.832,42.273,157.984
C02627=1035.305,174.211,-103.268,169.834,42.273,157.984
C02628=1035.311,174.460,-103.291,169.837,42.272,157.984
C02629=1035.317,174.709,-103.315,169.840,42.272,157.984
C02630=1035.323,174.958,-103.338,169.843,42.271,157.985
C02631=1035.329,175.207,-103.361,169.846,42.271,157.985
C02632=1035.335,175.456,-103.385,169.849,42.271,157.985
C02633=1035.342,175.704,-103.408,169.851,42.270,157.985
C02634=1035.347,175.953,-103.431,169.854,42.270,157.985
C02635=1035.353,176.202,-103.454,169.857,42.269,157.985
C02636=1035.360,176.451,-103.478,169.860,42.269,157.985
C02637=1035.366,176.700,-103.501,169.863,42.268,157.985
C02638=1035.372,176.949,-103.525,169.866,42.268,157.985
C02639=1035.379,177.197,-103.547,169.869,42.267,157.986
C02640=1035.385,177.446,-103.571,169.872,42.267,157.986
C02641=1035.391,177.695,-103.594,169.874,42.267,157.986
C02642=1035.397,177.944,-103.617,169.877,42.266,157.986
C02643=1035.403,178.192,-103.641,169.880,42.266,157.986
C02644=1035.409,178.442,-103.664,169.883,42.265,157.986
C02645=1035.415,178.690,-103.687,169.886,42.265,157.986
C02646=1035.422,178.940,-103.710,169.889,42.264,157.986
C02647=1035.428,179.188,-103.734,169.892,42.264,157.986
C02648=1035.434,179.437,-103.757,169.895,42.264,157.986
C02649=1035.441,179.686,-103.781,169.898,42.263,157.987
C02650=1035.446,179.935,-103.804,169.902,42.263,157.987
C02651=1035.453,180.184,-103.828,169.904,42.262,157.987
C02652=1035.459,180.433,-103.851,169.907,42.262,157.987
C02653=1035.465,180.681,-103.874,169.910,42.261,157.987
C02654=1035.472,180.929,-103.898,169.913,42.261,157.987
C02655=1035.478,181.178,-103.921,169.916,42.260,157.987
C02656=1035.485,181.427,-103.945,169.919,42.260,157.987
C02657=1035.490,181.676,-103.968,169.922,42.260,157.987
C02658=1035.497,181.925,-103.992,169.925,42.259,157.988
C02659=1035.503,182.173,-104.015,169.928,42.259,157.988
C02660=1035.509,182.423,-104.039,169.931,42.258,157.988
C02661=1035.515,182.671,-104.062,169.934,42.258,157.988
C02662=1035.523,182.920,-104.086,169.937,42.257,157.988
C02663=1035.528,183.169,-104.109,169.940,42.257,157.988
C02664=1035.534,183.418,-104.133,169.943,42.256,157.988
C02665=1035.540,183.666,-104.157,169.946,42.257,157.988
C02666=1035.546,183.916,-104.182,169.948,42.256,157.989
C02667=1035.552,184.164,-104.205,169.951,42.256,157.989
C02668=1035.558,184.413,-104.228,169.955,42.256,157.989
C02669=1035.564,184.662,-104.253,169.958,42.256,157.989
C02670=1035.570,184.910,-104.277,169.961,42.255,157.989
C02671=1035.576,185.160,-104.301,169.964,42.255,157.989
C02672=1035.582,185.408,-104.325,169.967,42.255,157.989
C02673=1035.587,185.657,-104.349,169.970,42.254,157.990
C02674=1035.594,185.906,-104.373,169.972,42.255,157.990
C02675=1035.599,186.154,-104.397,169.975,42.254,157.990
C02676=1035.606,186.403,-104.421,169.978,42.254,157.990
C02677=1035.611,186.652,-104.446,169.981,42.254,157.990
C02678=1035.618,186.901,-104.470,169.984,42.253,157.990
C02679=1035.624,187.149,-104.493,169.988,42.254,157.991
C02680=1035.630,187.398,-104.518,169.991,42.253,157.991
C02681=1035.636,187.647,-104.542,169.994,42.253,157.991
C02682=1035.642,187.896,-104.566,169.997,42.253,157.991
C02683=1035.648,188.144,-104.590,170.000,42.252,157.991
C02684=1035.653,188.393,-104.615,170.003,42.253,157.991
C02685=1035.660,188.678,-104.642,170.006,42.252,157.992
C02686=1035.667,188.962,-104.670,170.009,42.252,157.992
C02687=1035.674,189.245,-104.697,170.014,42.252,157.992
C02688=1035.681,189.529,-104.724,170.017,42.251,157.992
C02689=1035.687,189.778,-104.748,170.020,42.252,157.992
C02690=1035.693,190.028,-104.773,170.023,42.251,157.992
C02691=1035.699,190.275,-104.797,170.026,42.251,157.993
C02692=1035.705,190.525,-104.822,170.029,42.251,157.993
C02693=1035.711,190.773,-104.846,170.032,42.250,157.993
C02694=1035.717,191.022,-104.870,170.035,42.251,157.993
C02695=1035.723,191.271,-104.894,170.038,42.250,157.993
C02696=1035.729,191.520,-104.919,170.042,42.250,157.993
C02697=1035.736,191.768,-104.943,170.045,42.250,157.994
C02698=1035.741,192.017,-104.968,170.048,42.249,157.994
C02699=1035.748,192.266,-104.992,170.051,42.249,157.994
C02700=1035.753,192.514,-105.016,170.054,42.249,157.994
C02701=1035.760,192.763,-105.040,170.057,42.249,157.994
C02702=1035.766,193.012,-105.065,170.060,42.249,157.994
C02703=1035.772,193.260,-105.089,170.064,42.249,157.995
C02704=1035.778,193.510,-105.113,170.067,42.248,157.995
C02705=1035.785,193.759,-105.138,170.070,42.249,157.995
C02706=1035.790,194.006,-105.162,170.073,42.248,157.995
C02707=1035.797,194.255,-105.187,170.076,42.248,157.995
C02708=1035.803,194.505,-105.211,170.079,42.248,157.995
C02709=1035.808,194.753,-105.235,170.082,42.247,157.996
C02710=1035.815,195.002,-105.260,170.085,42.248,157.996
C02711=1035.821,195.251,-105.285,170.088,42.247,157.996
C02712=1035.827,195.499,-105.308,170.092,42.247,157.996
C02713=1035.833,195.748,-105.334,170.095,42.247,157.996
C02714=1035.840,195.997,-105.358,170.098,42.247,157.997
C02715=1035.846,196.246,-105.383,170.101,42.247,157.997
C02716=1035.852,196.494,-105.407,170.104,42.247,157.997
C02717=1035.858,196.743,-105.431,170.107,42.246,157.997
C02718=1035.865,196.992,-105.456,170.110,42.247,157.997
C02719=1035.870,197.240,-105.480,170.113,42.246,157.997
C02720=1035.877,197.488,-105.505,170.117,42.246,157.998
C02721=1035.883,197.738,-105.530,170.121,42.246,157.998
C02722=1035.890,197.987,-105.554,170.124,42.246,157.998
C02723=1035.896,198.235,-105.579,170.127,42.245,157.998
C02724=1035.902,198.484,-105.603,170.130,42.246,157.998
C02725=1035.908,198.732,-105.628,170.133,42.245,157.999
C02726=1035.914,198.982,-105.653,170.136,42.245,157.999
C02727=1035.921,199.230,-105.678,170.140,42.245,157.999
C02728=1035.927,199.479,-105.702,170.143,42.245,157.999
C02729=1035.933,199.727,-105.727,170.146,42.245,157.999
C02730=1035.939,199.976,-105.751,170.149,42.245,157.999
C02731=1035.946,200.225,-105.776,170.153,42.244,158.000
C02732=1035.952,200.474,-105.800,170.156,42.244,158.000
C02733=1035.959,200.722,-105.825,170.160,42.244,158.000
C02734=1035.965,200.970,-105.850,170.163,42.244,158.000
C02735=1035.971,201.219,-105.875,170.166,42.244,158.000
C02736=1035.977,201.468,-105.900,170.169,42.244,158.001
C02737=1035.983,201.717,-105.926,170.172,42.244,158.001
C02738=1035.989,201.966,-105.950,170.175,42.244,158.001
C02739=1035.995,202.215,-105.975,170.178,42.244,158.001
C02740=1036.001,202.463,-106.000,170.182,42.244,158.002
C02741=1036.007,202.711,-106.026,170.185,42.244,158.002
C02742=1036.014,202.960,-106.050,170.189,42.244,158.002
C02743=1036.020,203.209,-106.075,170.192,42.244,158.002
C02744=1036.026,203.458,-106.100,170.195,42.244,158.002
C02745=1036.032,203.706,-106.126,170.199,42.245,158.003
C02746=1036.037,203.955,-106.150,170.202,42.244,158.003
C02747=1036.044,204.204,-106.175,170.205,42.244,158.003
C02748=1036.050,204.452,-106.201,170.208,42.244,158.003
C02749=1036.076,205.502,-106.307,170.524,42.349,158.046
C02750=1036.086,205.832,-106.342,170.526,42.350,158.046
C02751=1036.094,206.162,-106.377,170.530,42.351,158.047
C02752=1036.103,206.491,-106.412,170.533,42.352,158.047
C02753=1036.112,206.821,-106.447,170.536,42.353,158.048
C02754=1036.119,207.069,-106.473,170.538,42.354,158.048
C02755=1036.125,207.318,-106.500,170.540,42.354,158.048
C02756=1036.132,207.566,-106.526,170.543,42.355,158.049
C02757=1036.139,207.815,-106.553,170.545,42.356,158.049
C02758=1036.146,208.063,-106.579,170.548,42.356,158.049
C02759=1036.152,208.312,-106.606,170.551,42.357,158.050
C02760=1036.159,208.560,-106.633,170.553,42.358,158.050
C02761=1036.166,208.808,-106.659,170.556,42.359,158.050
C02762=1036.173,209.057,-106.685,170.558,42.359,158.051
C02763=1036.179,209.306,-106.712,170.560,42.360,158.051
C02764=1036.186,209.554,-106.738,170.563,42.361,158.051
C02765=1036.193,209.803,-106.765,170.565,42.362,158.052
C02766=1036.199,210.051,-106.792,170.567,42.363,158.052
C02767=1036.206,210.300,-106.818,170.570,42.363,158.052
C02768=1036.213,210.549,-106.845,170.572,42.364,158.053
C02769=1036.219,210.797,-106.872,170.575,42.365,158.053
C02770=1036.226,211.045,-106.898,170.577,42.366,158.053
C02771=1036.233,211.294,-106.926,170.579,42.367,158.054
C02772=1036.239,211.542,-106.952,170.582,42.368,158.054
C02773=1036.246,211.791,-106.979,170.584,42.369,158.054
C02774=1036.253,212.039,-107.006,170.586,42.369,158.055
C02775=1036.259,212.287,-107.033,170.589,42.370,158.055
C02776=1036.266,212.536,-107.059,170.592,42.371,158.055
C02777=1036.273,212.785,-107.087,170.594,42.372,158.056
C02778=1036.279,213.033,-107.113,170.597,42.372,158.056
C02779=1036.286,213.282,-107.140,170.599,42.373,158.056
C02780=1036.293,213.530,-107.167,170.602,42.374,158.057
C02781=1036.299,213.778,-107.194,170.604,42.375,158.057
C02782=1036.306,214.027,-107.220,170.606,42.376,158.057
C02783=1036.313,214.275,-107.248,170.609,42.377,158.058
C02784=1036.320,214.524,-107.274,170.611,42.377,158.058
C02785=1036.326,214.772,-107.301,170.613,42.378,158.058
C02786=1036.333,215.021,-107.328,170.616,42.379,158.059
C02787=1036.339,215.270,-107.355,170.618,42.380,158.059
C02788=1036.346,215.517,-107.382,170.622,42.380,158.059
C02789=1036.353,215.766,-107.409,170.624,42.381,158.060
C02790=1036.360,216.014,-107.436,170.626,42.382,158.060
C02791=1036.366,216.263,-107.463,170.629,42.383,158.060
C02792=1036.372,216.511,-107.490,170.631,42.384,158.061
C02793=1036.380,216.760,-107.517,170.634,42.385,158.061
C02794=1036.386,217.008,-107.544,170.636,42.385,158.061
C02795=1036.393,217.257,-107.571,170.638,42.386,158.062
C02796=1036.400,217.506,-107.598,170.642,42.387,158.062
C02797=1036.407,217.754,-107.625,170.644,42.388,158.062
C02798=1036.413,218.002,-107.652,170.646,42.388,158.063
C02799=1036.420,218.251,-107.679,170.649,42.389,158.063
C02800=1036.427,218.499,-107.706,170.651,42.390,158.063
C02801=1036.434,218.748,-107.733,170.653,42.391,158.064
C02802=1036.440,218.996,-107.760,170.657,42.391,158.064
C02803=1036.447,219.245,-107.787,170.659,42.392,158.064
C02804=1036.454,219.493,-107.814,170.662,42.393,158.065
C02805=1036.461,219.741,-107.842,170.664,42.394,158.065
C02806=1036.469,220.077,-107.878,170.668,42.395,158.066
C02807=1036.479,220.412,-107.915,170.671,42.396,158.066
C02808=1036.488,220.747,-107.952,170.675,42.397,158.067
C02809=1036.497,221.082,-107.989,170.678,42.399,158.067
C02810=1036.503,221.331,-108.016,170.680,42.399,158.067
C02811=1036.509,221.579,-108.044,170.683,42.400,158.068
C02812=1036.516,221.827,-108.071,170.685,42.401,158.068
C02813=1036.523,222.076,-108.099,170.688,42.402,158.068
C02814=1036.530,222.325,-108.125,170.690,42.403,158.069
C02815=1036.537,222.573,-108.153,170.694,42.404,158.069
C02816=1036.543,222.821,-108.180,170.696,42.404,158.069
C02817=1036.549,223.069,-108.208,170.698,42.405,158.070
C02818=1036.556,223.318,-108.235,170.701,42.406,158.070
C02819=1036.562,223.567,-108.263,170.703,42.407,158.070
C02820=1036.570,223.815,-108.290,170.706,42.407,158.071
C02821=1036.577,224.063,-108.318,170.709,42.408,158.071
C02822=1036.583,224.312,-108.346,170.711,42.409,158.072
C02823=1036.590,224.560,-108.373,170.714,42.410,158.072
C02824=1036.596,224.809,-108.400,170.716,42.411,158.072
C02825=1036.602,225.057,-108.428,170.720,42.412,158.073
C02826=1036.610,225.305,-108.455,170.722,42.413,158.073
C02827=1036.616,225.554,-108.483,170.724,42.414,158.073
C02828=1036.623,225.802,-108.510,170.727,42.414,158.074
C02829=1036.630,226.050,-108.538,170.729,42.415,158.074
C02830=1036.637,226.299,-108.566,170.732,42.416,158.074
C02831=1036.643,226.547,-108.593,170.735,42.417,158.075
C02832=1036.651,226.795,-108.621,170.737,42.418,158.075
C02833=1036.657,227.044,-108.648,170.740,42.419,158.075
C02834=1036.664,227.293,-108.675,170.743,42.419,158.076
C02835=1036.670,227.541,-108.703,170.746,42.420,158.076
C02836=1036.677,227.790,-108.731,170.748,42.421,158.077
C02837=1036.684,228.038,-108.759,170.750,42.422,158.077
C02838=1036.690,228.287,-108.786,170.754,42.422,158.077
C02839=1036.697,228.535,-108.814,170.756,42.423,158.078
C02840=1036.704,228.784,-108.842,170.758,42.424,158.078
C02841=1036.710,229.031,-108.870,170.761,42.425,158.078
C02842=1036.717,229.279,-108.898,170.764,42.426,158.079
C02843=1036.723,229.528,-108.925,170.767,42.427,158.079
C02844=1036.730,229.776,-108.953,170.769,42.428,158.079
C02845=1036.737,230.024,-108.981,170.772,42.429,158.080
C02846=1036.744,230.273,-109.008,170.775,42.430,158.080
C02847=1036.750,230.521,-109.036,170.777,42.430,158.081
C02848=1036.757,230.770,-109.064,170.780,42.431,158.081
C02849=1036.763,231.018,-109.093,170.782,42.432,158.081
C02850=1036.770,231.266,-109.121,170.786,42.433,158.082
C02851=1036.777,231.515,-109.148,170.788,42.434,158.082
C02852=1036.783,231.763,-109.176,170.790,42.435,158.082
C02853=1036.790,232.012,-109.204,170.794,42.436,158.083
C02854=1036.797,232.260,-109.232,170.796,42.437,158.083
C02855=1036.804,232.508,-109.260,170.799,42.438,158.084
C02856=1036.809,232.757,-109.288,170.801,42.439,158.084
C02857=1036.816,233.005,-109.316,170.805,42.439,158.084
C02858=1036.823,233.253,-109.345,170.807,42.440,158.085
C02859=1036.830,233.501,-109.372,170.810,42.442,158.085
C02860=1036.836,233.750,-109.401,170.813,42.443,158.086
C02861=1036.843,233.998,-109.429,170.815,42.444,158.086
C02862=1036.851,234.326,-109.466,170.819,42.444,158.086
C02863=1036.861,234.654,-109.503,170.823,42.446,158.087
C02864=1036.869,234.982,-109.540,170.826,42.447,158.087
C02865=1036.878,235.309,-109.577,170.830,42.448,158.088
C02866=1036.885,235.558,-109.605,170.832,42.449,158.088
C02867=1036.891,235.806,-109.634,170.835,42.450,158.089
C02868=1036.898,236.054,-109.662,170.838,42.451,158.089
C02869=1036.905,236.302,-109.690,170.840,42.452,158.090
C02870=1036.912,236.551,-109.718,170.844,42.453,158.090
C02871=1036.917,236.799,-109.746,170.846,42.454,158.090
C02872=1036.924,237.047,-109.775,170.849,42.455,158.091
C02873=1036.932,237.296,-109.803,170.852,42.455,158.091
C02874=1036.939,237.544,-109.831,170.855,42.456,158.091
C02875=1036.945,237.793,-109.860,170.857,42.457,158.092
C02876=1036.952,238.041,-109.888,170.860,42.458,158.092
C02877=1036.958,238.289,-109.916,170.863,42.459,158.093
C02878=1036.965,238.537,-109.944,170.865,42.460,158.093
C02879=1036.971,238.786,-109.972,170.869,42.461,158.093
C02880=1036.979,239.034,-110.001,170.871,42.462,158.094
C02881=1036.986,239.283,-110.029,170.875,42.462,158.094
C02882=1036.992,239.531,-110.058,170.877,42.463,158.094
C02883=1036.998,239.779,-110.086,170.879,42.464,158.095
C02884=1037.005,240.027,-110.114,170.883,42.466,158.095
C02885=1037.012,240.275,-110.143,170.885,42.467,158.096
C02886=1037.019,240.524,-110.171,170.888,42.468,158.096
C02887=1037.026,240.772,-110.200,170.891,42.468,158.097
C02888=1037.032,241.020,-110.229,170.894,42.469,158.097
C02889=1037.039,241.269,-110.257,170.897,42.470,158.097
C02890=1037.045,241.517,-110.286,170.900,42.471,158.098
C02891=1037.051,241.765,-110.315,170.902,42.472,158.098
C02892=1037.059,242.014,-110.343,170.906,42.473,158.099
C02893=1037.065,242.262,-110.372,170.908,42.474,158.099
C02894=1037.072,242.510,-110.400,170.910,42.475,158.099
C02895=1037.078,242.758,-110.429,170.914,42.476,158.100
C02896=1037.085,243.007,-110.457,170.916,42.477,158.100
C02897=1037.092,243.256,-110.486,170.920,42.478,158.101
C02898=1037.098,243.504,-110.515,170.922,42.479,158.101
C02899=1037.105,243.752,-110.544,170.925,42.480,158.101
C02900=1037.111,244.000,-110.573,170.928,42.481,158.102
C02901=1037.118,244.248,-110.601,170.931,42.482,158.102
C02902=1037.125,244.497,-110.630,170.934,42.483,158.103
C02903=1037.132,244.745,-110.659,170.937,42.484,158.103
C02904=1037.138,244.993,-110.688,170.939,42.485,158.103
C02905=1037.144,245.241,-110.717,170.943,42.486,158.104
C02906=1037.150,245.489,-110.746,170.945,42.487,158.104
C02907=1037.157,245.738,-110.775,170.949,42.488,158.105
C02908=1037.164,245.986,-110.804,170.951,42.489,158.105
C02909=1037.171,246.234,-110.833,170.954,42.491,158.106
C02910=1037.177,246.482,-110.862,170.957,42.491,158.106
C02911=1037.184,246.731,-110.891,170.959,42.492,158.106
C02912=1037.190,246.979,-110.920,170.963,42.494,158.107
C02913=1037.196,247.227,-110.949,170.966,42.495,158.107
C02914=1037.203,247.475,-110.978,170.969,42.495,158.108
C02915=1037.210,247.724,-111.007,170.971,42.496,158.108
C02916=1037.216,247.972,-111.036,170.974,42.498,158.109
C02917=1037.222,248.220,-111.065,170.977,42.498,158.109
C02918=1037.231,248.542,-111.103,170.981,42.500,158.109
C02919=1037.240,248.864,-111.140,170.985,42.501,158.110
C02920=1037.248,249.186,-111.178,170.988,42.503,158.111
C02921=1037.257,249.507,-111.216,170.993,42.504,158.111
C02922=1037.264,249.756,-111.246,170.996,42.505,158.112
C02923=1037.270,250.004,-111.275,170.998,42.506,158.112
C02924=1037.276,250.252,-111.304,171.001,42.507,158.112
C02925=1037.283,250.500,-111.332,171.004,42.508,158.113
C02926=1037.290,250.749,-111.361,171.007,42.509,158.113
C02927=1037.296,250.996,-111.391,171.010,42.510,158.114
C02928=1037.303,251.245,-111.421,171.013,42.511,158.114
C02929=1037.310,251.493,-111.450,171.016,42.513,158.115
C02930=1037.316,251.742,-111.479,171.019,42.513,158.115
C02931=1037.323,251.990,-111.509,171.022,42.514,158.115
C02932=1037.330,252.238,-111.537,171.025,42.516,158.116
C02933=1037.336,252.486,-111.566,171.028,42.517,158.116
C02934=1037.343,252.735,-111.596,171.032,42.518,158.117
C02935=1037.350,252.982,-111.625,171.034,42.519,158.117
C02936=1037.356,253.231,-111.655,171.037,42.520,158.118
C02937=1037.363,253.479,-111.684,171.040,42.521,158.118
C02938=1037.369,253.727,-111.713,171.043,42.522,158.119
C02939=1037.376,253.975,-111.743,171.046,42.523,158.119
C02940=1037.383,254.223,-111.772,171.049,42.524,158.120
C02941=1037.390,254.472,-111.801,171.053,42.525,158.120
C02942=1037.396,254.720,-111.831,171.055,42.526,158.120
C02943=1037.403,254.968,-111.860,171.059,42.527,158.121
C02944=1037.410,255.216,-111.890,171.061,42.528,158.121
C02945=1037.417,255.465,-111.919,171.065,42.529,158.122
C02946=1037.423,255.713,-111.948,171.067,42.531,158.122
C02947=1037.430,255.960,-111.978,171.071,42.531,158.123
C02948=1037.437,256.209,-112.007,171.073,42.532,158.123
C02949=1037.444,256.456,-112.037,171.077,42.534,158.123
C02950=1037.451,256.705,-112.066,171.080,42.534,158.124
C02951=1037.457,256.953,-112.095,171.083,42.536,158.124
C02952=1037.464,257.202,-112.125,171.086,42.537,158.125
C02953=1037.470,257.450,-112.154,171.089,42.538,158.125
C02954=1037.477,257.698,-112.184,171.092,42.539,158.126
C02955=1037.484,257.947,-112.214,171.095,42.540,158.126
C02956=1037.491,258.194,-112.244,171.098,42.541,158.126
C02957=1037.498,258.443,-112.273,171.102,42.542,158.127
C02958=1037.505,258.690,-112.302,171.104,42.543,158.127
C02959=1037.512,258.939,-112.332,171.108,42.544,158.128
C02960=1037.518,259.187,-112.361,171.111,42.545,158.128
C02961=1037.525,259.435,-112.391,171.114,42.546,158.129
C02962=1037.532,259.683,-112.420,171.118,42.547,158.129
C02963=1037.539,259.931,-112.451,171.120,42.548,158.130
C02964=1037.546,260.180,-112.480,171.123,42.549,158.130
C02965=1037.552,260.428,-112.510,171.127,42.550,158.131
C02966=1037.559,260.676,-112.540,171.129,42.551,158.131
C02967=1037.566,260.924,-112.569,171.133,42.553,158.132
C02968=1037.573,261.172,-112.599,171.136,42.553,158.132
C02969=1037.581,261.420,-112.629,171.139,42.554,158.132
C02970=1037.587,261.668,-112.658,171.143,42.556,158.133
C02971=1037.594,261.916,-112.688,171.146,42.556,158.133
C02972=1037.601,262.165,-112.718,171.149,42.558,158.134
C02973=1037.607,262.412,-112.748,171.152,42.559,158.134
C02974=1037.616,262.733,-112.787,171.156,42.561,158.135
C02975=1037.624,263.054,-112.825,171.161,42.562,158.135
C02976=1037.632,263.374,-112.865,171.164,42.564,158.136
C02977=1037.641,263.695,-112.903,171.168,42.565,158.137
C02978=1037.648,263.942,-112.933,171.171,42.566,158.137
C02979=1037.655,264.190,-112.963,171.175,42.567,158.138
C02980=1037.661,264.439,-112.994,171.178,42.569,158.138
C02981=1037.668,264.686,-113.024,171.181,42.570,158.139
C02982=1037.675,264.935,-113.054,171.185,42.571,158.139
C02983=1037.682,265.183,-113.083,171.187,42.572,158.140
C02984=1037.688,265.431,-113.114,171.191,42.573,158.140
C02985=1037.695,265.679,-113.144,171.194,42.575,158.141
C02986=1037.702,265.928,-113.174,171.197,42.575,158.141
C02987=1037.708,266.176,-113.204,171.201,42.577,158.142
C02988=1037.715,266.424,-113.234,171.204,42.578,158.142
C02989=1037.722,266.672,-113.264,171.207,42.579,158.142
C02990=1037.728,266.920,-113.295,171.210,42.580,158.143
C02991=1037.735,267.167,-113.326,171.214,42.581,158.143
C02992=1037.743,267.416,-113.356,171.216,42.583,158.144
C02993=1037.748,267.663,-113.386,171.220,42.584,158.144
C02994=1037.756,267.912,-113.416,171.223,42.585,158.145
C02995=1037.762,268.160,-113.447,171.226,42.586,158.145
C02996=1037.769,268.408,-113.477,171.230,42.588,158.146
C02997=1037.775,268.656,-113.507,171.233,42.588,158.146
C02998=1037.782,268.904,-113.538,171.236,42.590,158.147
C02999=1037.789,269.152,-113.569,171.239,42.591,158.147
C03000=1037.795,269.400,-113.599,171.243,42.593,158.148
C03001=1037.803,269.648,-113.629,171.246,42.593,158.148
C03002=1037.809,269.897,-113.660,171.249,42.595,158.149
C03003=1037.816,270.144,-113.690,171.253,42.596,158.149
C03004=1037.822,270.392,-113.721,171.256,42.597,158.150
C03005=1037.829,270.640,-113.751,171.259,42.599,158.150
C03006=1037.836,270.889,-113.782,171.262,42.600,158.151
C03007=1037.843,271.136,-113.812,171.266,42.601,158.152
C03008=1037.849,271.384,-113.843,171.269,42.602,158.152
C03009=1037.856,271.633,-113.874,171.272,42.604,158.152
C03010=1037.863,271.880,-113.904,171.276,42.605,158.153
C03011=1037.869,272.129,-113.935,171.279,42.606,158.154
C03012=1037.877,272.377,-113.965,171.283,42.608,158.154
C03013=1037.883,272.624,-113.996,171.285,42.609,158.154
C03014=1037.889,272.873,-114.027,171.289,42.610,158.155
C03015=1037.897,273.120,-114.058,171.293,42.611,158.156
C03016=1037.903,273.369,-114.089,171.296,42.613,158.156
C03017=1037.910,273.617,-114.120,171.299,42.614,158.157
C03018=1037.916,273.864,-114.150,171.303,42.616,158.157
C03019=1037.923,274.113,-114.180,171.306,42.616,158.158
C03020=1037.930,274.360,-114.211,171.310,42.618,158.158
C03021=1037.937,274.609,-114.242,171.312,42.619,158.159
C03022=1037.943,274.857,-114.273,171.316,42.621,158.159
C03023=1037.950,275.105,-114.305,171.320,42.622,158.160
C03024=1037.957,275.352,-114.335,171.323,42.623,158.160
C03025=1037.963,275.600,-114.366,171.327,42.625,158.161
C03026=1037.970,275.849,-114.397,171.329,42.625,158.161
C03027=1037.976,276.096,-114.428,171.333,42.627,158.162
C03028=1037.984,276.344,-114.459,171.337,42.628,158.162
C03029=1037.990,276.593,-114.490,171.340,42.630,158.163
C03030=1037.999,276.917,-114.530,171.344,42.631,158.164
C03031=1038.008,277.242,-114.571,171.349,42.633,158.164
C03032=1038.017,277.568,-114.612,171.354,42.635,158.165
C03033=1038.026,277.893,-114.652,171.358,42.636,158.166
C03034=1038.032,278.141,-114.683,171.361,42.638,158.166
C03035=1038.040,278.388,-114.714,171.365,42.639,158.167
C03036=1038.046,278.636,-114.746,171.368,42.640,158.167
C03037=1038.053,278.885,-114.776,171.372,42.642,158.168
C03038=1038.060,279.133,-114.808,171.376,42.643,158.169
C03039=1038.066,279.381,-114.839,171.378,42.645,158.169
C03040=1038.073,279.628,-114.871,171.382,42.646,158.170
C03041=1038.080,279.876,-114.902,171.386,42.647,158.170
C03042=1038.086,280.124,-114.933,171.389,42.649,158.171
C03043=1038.093,280.371,-114.965,171.393,42.650,158.171
C03044=1038.099,280.619,-114.996,171.397,42.652,158.172
C03045=1038.106,280.868,-115.027,171.399,42.654,158.172
C03046=1038.112,281.116,-115.058,171.403,42.655,158.173
C03047=1038.119,281.364,-115.090,171.407,42.656,158.174
C03048=1038.126,281.612,-115.121,171.410,42.658,158.174
C03049=1038.133,281.859,-115.153,171.414,42.659,158.175
C03050=1038.139,282.107,-115.184,171.418,42.660,158.175
C03051=1038.146,282.355,-115.215,171.421,42.662,158.176
C03052=1038.153,282.603,-115.247,171.424,42.663,158.176
C03053=1038.160,282.851,-115.278,171.427,42.665,158.177
C03054=1038.166,283.099,-115.310,171.431,42.666,158.177
C03055=1038.173,283.347,-115.341,171.435,42.667,158.178
C03056=1038.180,283.595,-115.373,171.438,42.669,158.179
C03057=1038.187,283.843,-115.404,171.442,42.670,158.179
C03058=1038.194,284.091,-115.436,171.446,42.672,158.180
C03059=1038.201,284.339,-115.468,171.450,42.673,158.180
C03060=1038.208,284.586,-115.499,171.453,42.675,158.181
C03061=1038.214,284.834,-115.531,171.457,42.676,158.182
C03062=1038.221,285.082,-115.562,171.460,42.677,158.182
C03063=1038.228,285.330,-115.594,171.463,42.679,158.183
C03064=1038.234,285.578,-115.625,171.467,42.680,158.183
C03065=1038.241,285.825,-115.657,171.471,42.682,158.184
C03066=1038.248,286.073,-115.689,171.474,42.683,158.184
C03067=1038.256,286.322,-115.720,171.478,42.685,158.185
C03068=1038.262,286.570,-115.752,171.482,42.686,158.186
C03069=1038.269,286.818,-115.783,171.485,42.687,158.186
C03070=1038.276,287.065,-115.815,171.489,42.689,158.187
C03071=1038.283,287.313,-115.847,171.493,42.691,158.187
C03072=1038.289,287.561,-115.878,171.496,42.692,158.188
C03073=1038.296,287.808,-115.911,171.500,42.693,158.189
C03074=1038.302,288.056,-115.943,171.504,42.695,158.189
C03075=1038.310,288.305,-115.974,171.507,42.697,158.190
C03076=1038.317,288.552,-116.006,171.511,42.698,158.190
C03077=1038.324,288.800,-116.038,171.515,42.699,158.191
C03078=1038.330,289.048,-116.071,171.519,42.701,158.192
C03079=1038.337,289.296,-116.102,171.522,42.703,158.192
C03080=1038.344,289.544,-116.135,171.526,42.704,158.193
C03081=1038.351,289.791,-116.166,171.530,42.706,158.193
C03082=1038.357,290.039,-116.199,171.533,42.707,158.194
C03083=1038.364,290.287,-116.230,171.536,42.709,158.195
C03084=1038.371,290.534,-116.262,171.540,42.711,158.195
C03085=1038.378,290.783,-116.295,171.544,42.712,158.196
C03086=1038.387,291.119,-116.338,171.550,42.714,158.197
C03087=1038.396,291.457,-116.382,171.554,42.716,158.197
C03088=1038.406,291.794,-116.425,171.560,42.718,158.198
C03089=1038.414,292.130,-116.469,171.564,42.720,158.199
C03090=1038.421,292.378,-116.501,171.568,42.722,158.200
C03091=1038.429,292.626,-116.533,171.572,42.723,158.200
C03092=1038.435,292.874,-116.566,171.576,42.725,158.201
C03093=1038.442,293.122,-116.598,171.579,42.727,158.202
C03094=1038.449,293.370,-116.630,171.583,42.728,158.202
C03095=1038.456,293.617,-116.663,171.587,42.730,158.203
C03096=1038.463,293.865,-116.695,171.591,42.731,158.204
C03097=1038.469,294.113,-116.727,171.594,42.733,158.204
C03098=1038.476,294.361,-116.759,171.598,42.735,158.205
C03099=1038.483,294.608,-116.792,171.602,42.737,158.205
C03100=1038.490,294.856,-116.824,171.606,42.738,158.206
C03101=1038.497,295.104,-116.856,171.609,42.740,158.207
C03102=1038.503,295.352,-116.889,171.613,42.741,158.207
C03103=1038.510,295.599,-116.922,171.617,42.743,158.208
C03104=1038.517,295.847,-116.954,171.621,42.745,158.209
C03105=1038.524,296.095,-116.987,171.624,42.746,158.209
C03106=1038.530,296.343,-117.020,171.628,42.748,158.210
C03107=1038.536,296.590,-117.052,171.632,42.750,158.211
C03108=1038.544,296.838,-117.085,171.636,42.752,158.211
C03109=1038.550,297.086,-117.118,171.640,42.753,158.212
C03110=1038.556,297.333,-117.150,171.645,42.755,158.213
C03111=1038.563,297.582,-117.184,171.648,42.757,158.213
C03112=1038.570,297.829,-117.216,171.652,42.758,158.214
C03113=1038.577,298.077,-117.248,171.656,42.760,158.215
C03114=1038.584,298.324,-117.282,171.660,42.762,158.215
C03115=1038.590,298.572,-117.315,171.663,42.764,158.216
C03116=1038.597,298.819,-117.347,171.667,42.766,158.217
C03117=1038.604,299.067,-117.380,171.671,42.768,158.217
C03118=1038.610,299.315,-117.413,171.675,42.769,158.218
C03119=1038.617,299.563,-117.446,171.679,42.771,158.219
C03120=1038.624,299.810,-117.480,171.683,42.773,158.219
C03121=1038.631,300.058,-117.512,171.686,42.774,158.220
C03122=1038.638,300.306,-117.545,171.691,42.776,158.221
C03123=1038.644,300.553,-117.578,171.695,42.778,158.221
C03124=1038.651,300.802,-117.611,171.699,42.780,158.222
C03125=1038.658,301.048,-117.644,171.703,42.782,158.223
C03126=1038.665,301.297,-117.677,171.706,42.783,158.223
C03127=1038.671,301.544,-117.709,171.710,42.785,158.224
C03128=1038.679,301.792,-117.743,171.714,42.787,158.225
C03129=1038.685,302.039,-117.776,171.718,42.789,158.226
C03130=1038.693,302.287,-117.808,171.723,42.790,158.226
C03131=1038.699,302.534,-117.842,171.726,42.792,158.227
C03132=1038.706,302.783,-117.875,171.730,42.794,158.228
C03133=1038.712,303.030,-117.908,171.734,42.796,158.228
C03134=1038.720,303.278,-117.942,171.738,42.798,158.229
C03135=1038.727,303.525,-117.974,171.742,42.799,158.230
C03136=1038.734,303.773,-118.008,171.746,42.801,158.230
C03137=1038.740,304.021,-118.040,171.750,42.803,158.231
C03138=1038.747,304.269,-118.073,171.754,42.804,158.232
C03139=1038.754,304.517,-118.107,171.758,42.806,158.233
C03140=1038.761,304.764,-118.139,171.762,42.808,158.233
C03141=1038.768,305.011,-118.173,171.767,42.810,158.234
C03142=1038.778,305.365,-118.221,171.772,42.812,158.235
C03143=1038.788,305.719,-118.268,171.778,42.815,158.236
C03144=1038.798,306.073,-118.316,171.783,42.818,158.237
C03145=1038.808,306.426,-118.363,171.790,42.820,158.238
C03146=1038.815,306.674,-118.396,171.793,42.822,158.239
C03147=1038.822,306.921,-118.430,171.797,42.824,158.239
C03148=1038.829,307.169,-118.463,171.802,42.826,158.240
C03149=1038.836,307.417,-118.497,171.806,42.828,158.241
C03150=1038.843,307.663,-118.530,171.810,42.830,158.242
C03151=1038.850,307.912,-118.563,171.814,42.832,158.242
C03152=1038.857,308.159,-118.597,171.819,42.833,158.243
C03153=1038.865,308.407,-118.630,171.823,42.835,158.244
C03154=1038.871,308.655,-118.663,171.826,42.837,158.245
C03155=1038.878,308.902,-118.697,171.831,42.839,158.245
C03156=1038.885,309.150,-118.731,171.835,42.841,158.246
C03157=1038.893,309.397,-118.764,171.839,42.843,158.247
C03158=1038.899,309.645,-118.797,171.843,42.845,158.247
C03159=1038.907,309.893,-118.831,171.848,42.846,158.248
C03160=1038.914,310.140,-118.864,171.852,42.848,158.249
C03161=1038.921,310.388,-118.898,171.855,42.850,158.250
C03162=1038.928,310.636,-118.932,171.860,42.852,158.250
C03163=1038.936,310.882,-118.965,171.864,42.854,158.251
C03164=1038.942,311.131,-118.998,171.868,42.856,158.252
C03165=1038.950,311.378,-119.032,171.873,42.858,158.253
C03166=1038.957,311.626,-119.066,171.877,42.860,158.253
C03167=1038.964,311.874,-119.099,171.881,42.861,158.254
C03168=1038.971,312.121,-119.133,171.886,42.863,158.255
C03169=1038.978,312.368,-119.167,171.890,42.866,158.256
C03170=1038.984,312.616,-119.201,171.894,42.868,158.256
C03171=1038.992,312.863,-119.236,171.899,42.870,158.257
C03172=1038.998,313.111,-119.270,171.902,42.872,158.258
C03173=1039.005,313.358,-119.304,171.906,42.874,158.259
C03174=1039.011,313.606,-119.338,171.910,42.876,158.260
C03175=1039.019,313.854,-119.372,171.915,42.878,158.260
C03176=1039.026,314.101,-119.406,171.919,42.880,158.261
C03177=1039.033,314.349,-119.441,171.923,42.882,158.262
C03178=1039.039,314.596,-119.474,171.928,42.884,158.263
C03179=1039.046,314.844,-119.509,171.932,42.887,158.264
C03180=1039.053,315.091,-119.543,171.936,42.889,158.264
C03181=1039.060,315.339,-119.578,171.941,42.890,158.265
C03182=1039.067,315.587,-119.611,171.945,42.893,158.266
C03183=1039.074,315.834,-119.647,171.949,42.895,158.267
C03184=1039.081,316.082,-119.680,171.954,42.897,158.268
C03185=1039.087,316.330,-119.715,171.958,42.899,158.268
C03186=1039.094,316.576,-119.749,171.962,42.901,158.269
C03187=1039.101,316.824,-119.783,171.967,42.903,158.270
C03188=1039.108,317.071,-119.818,171.971,42.906,158.271
C03189=1039.115,317.319,-119.852,171.976,42.907,158.272
C03190=1039.122,317.566,-119.887,171.980,42.910,158.273
C03191=1039.129,317.814,-119.921,171.984,42.912,158.273
C03192=1039.136,318.061,-119.956,171.989,42.914,158.274
C03193=1039.143,318.309,-119.990,171.993,42.916,158.275
C03194=1039.150,318.556,-120.025,171.998,42.918,158.276
C03195=1039.157,318.804,-120.059,172.002,42.920,158.277
C03196=1039.164,319.051,-120.094,172.006,42.923,158.277
C03197=1039.171,319.299,-120.128,172.011,42.925,158.278
C03198=1039.181,319.658,-120.178,172.017,42.928,158.279
C03199=1039.191,320.016,-120.228,172.024,42.931,158.281
C03200=1039.202,320.374,-120.278,172.030,42.935,158.282
C03201=1039.212,320.733,-120.329,172.037,42.937,158.283
C03202=1039.220,320.980,-120.363,172.041,42.940,158.284
C03203=1039.226,321.228,-120.398,172.046,42.942,158.285
C03204=1039.234,321.475,-120.432,172.050,42.944,158.286
C03205=1039.240,321.723,-120.467,172.055,42.946,158.286
C03206=1039.248,321.970,-120.501,172.059,42.949,158.287
C03207=1039.255,322.217,-120.537,172.064,42.951,158.288
C03208=1039.263,322.465,-120.571,172.068,42.953,158.289
C03209=1039.269,322.712,-120.607,172.073,42.955,158.290
C03210=1039.277,322.960,-120.640,172.077,42.957,158.291
C03211=1039.283,323.207,-120.676,172.082,42.960,158.292
C03212=1039.291,323.454,-120.710,172.086,42.962,158.292
C03213=1039.298,323.702,-120.746,172.091,42.964,158.293
C03214=1039.305,323.950,-120.781,172.095,42.966,158.294
C03215=1039.313,324.197,-120.815,172.100,42.969,158.295
C03216=1039.319,324.444,-120.850,172.104,42.971,158.296
C03217=1039.327,324.693,-120.885,172.109,42.973,158.297
C03218=1039.334,324.940,-120.920,172.113,42.976,158.298
C03219=1039.341,325.187,-120.954,172.118,42.978,158.298
C03220=1039.348,325.434,-120.989,172.122,42.980,158.299
C03221=1039.356,325.682,-121.024,172.127,42.982,158.300
C03222=1039.363,325.929,-121.059,172.132,42.985,158.301
C03223=1039.371,326.176,-121.094,172.137,42.987,158.302
C03224=1039.378,326.425,-121.129,172.142,42.989,158.303
C03225=1039.385,326.671,-121.165,172.146,42.991,158.304
C03226=1039.393,326.918,-121.200,172.151,42.994,158.305
C03227=1039.400,327.166,-121.235,172.155,42.996,158.305
C03228=1039.407,327.413,-121.270,172.160,42.998,158.306
C03229=1039.415,327.662,-121.305,172.165,43.001,158.307
C03230=1039.422,327.909,-121.340,172.169,43.003,158.308
C03231=1039.429,328.156,-121.375,172.174,43.005,158.309
C03232=1039.437,328.404,-121.410,172.178,43.008,158.310
C03233=1039.444,328.650,-121.446,172.183,43.010,158.311
C03234=1039.452,328.899,-121.481,172.189,43.013,158.312
C03235=1039.458,329.146,-121.516,172.193,43.015,158.313
C03236=1039.465,329.393,-121.552,172.198,43.017,158.314
C03237=1039.473,329.641,-121.588,172.202,43.020,158.315
C03238=1039.480,329.887,-121.624,172.207,43.022,158.315
C03239=1039.487,330.136,-121.659,172.212,43.025,158.317
C03240=1039.494,330.383,-121.694,172.216,43.027,158.317
C03241=1039.501,330.630,-121.730,172.221,43.030,158.318
C03242=1039.508,330.878,-121.766,172.227,43.032,158.319
C03243=1039.516,331.124,-121.802,172.231,43.035,158.320
C03244=1039.523,331.372,-121.837,172.236,43.037,158.321
C03245=1039.531,331.619,-121.872,172.240,43.040,158.322
C03246=1039.538,331.867,-121.908,172.245,43.042,158.323
C03247=1039.545,332.114,-121.944,172.250,43.044,158.324
C03248=1039.553,332.361,-121.980,172.255,43.048,158.325
C03249=1039.560,332.609,-122.015,172.260,43.050,158.326
C03250=1039.567,332.856,-122.051,172.265,43.052,158.327
C03251=1039.574,333.103,-122.087,172.269,43.055,158.328
C03252=1039.582,333.351,-122.123,172.274,43.057,158.329
C03253=1039.589,333.598,-122.158,172.279,43.060,158.330
C03254=1039.599,333.952,-122.210,172.286,43.064,158.331
C03255=1039.610,334.305,-122.261,172.293,43.068,158.333
C03256=1039.620,334.659,-122.313,172.301,43.071,158.334
C03257=1039.631,335.013,-122.364,172.307,43.075,158.335
C03258=1039.638,335.260,-122.400,172.313,43.077,158.336
C03259=1039.646,335.507,-122.436,172.318,43.080,158.337
C03260=1039.652,335.754,-122.473,172.322,43.083,158.338
C03261=1039.660,336.002,-122.509,172.327,43.085,158.339
C03262=1039.667,336.249,-122.545,172.333,43.088,158.340
C03263=1039.674,336.496,-122.581,172.337,43.090,158.341
C03264=1039.681,336.743,-122.618,172.342,43.093,158.342
C03265=1039.689,336.991,-122.654,172.347,43.096,158.343
C03266=1039.696,337.238,-122.690,172.352,43.098,158.344
C03267=1039.704,337.485,-122.726,172.357,43.102,158.345
C03268=1039.711,337.733,-122.763,172.362,43.104,158.346
C03269=1039.718,337.980,-122.799,172.367,43.107,158.347
C03270=1039.726,338.227,-122.835,172.373,43.110,158.349
C03271=1039.733,338.474,-122.871,172.378,43.112,158.349
C03272=1039.740,338.722,-122.908,172.382,43.115,158.351
C03273=1039.747,338.969,-122.944,172.387,43.118,158.352
C03274=1039.755,339.216,-122.980,172.392,43.120,158.353
C03275=1039.762,339.464,-123.017,172.398,43.123,158.354
C03276=1039.770,339.711,-123.054,172.403,43.126,158.355
C03277=1039.777,339.958,-123.089,172.407,43.129,158.356
C03278=1039.785,340.205,-123.126,172.413,43.131,158.357
C03279=1039.792,340.452,-123.163,172.418,43.134,158.358
C03280=1039.799,340.700,-123.199,172.423,43.137,158.359
C03281=1039.807,340.947,-123.236,172.429,43.140,158.360
C03282=1039.815,341.193,-123.272,172.434,43.142,158.361
C03283=1039.821,341.441,-123.309,172.438,43.145,158.362
C03284=1039.829,341.689,-123.345,172.443,43.148,158.363
C03285=1039.836,341.936,-123.383,172.449,43.151,158.364
C03286=1039.844,342.183,-123.419,172.454,43.154,158.365
C03287=1039.851,342.430,-123.457,172.459,43.156,158.366
C03288=1039.859,342.678,-123.493,172.465,43.159,158.367
C03289=1039.866,342.924,-123.530,172.470,43.162,158.368
C03290=1039.873,343.172,-123.566,172.474,43.165,158.369
C03291=1039.881,343.419,-123.604,172.480,43.168,158.371
C03292=1039.889,343.666,-123.641,172.485,43.171,158.372
C03293=1039.895,343.913,-123.677,172.490,43.174,158.373
C03294=1039.903,344.160,-123.714,172.496,43.177,158.374
C03295=1039.911,344.407,-123.752,172.501,43.179,158.375
C03296=1039.918,344.655,-123.788,172.507,43.183,158.376
C03297=1039.926,344.902,-123.826,172.512,43.186,158.377
C03298=1039.934,345.149,-123.863,172.517,43.189,158.378
C03299=1039.941,345.396,-123.899,172.523,43.191,158.379
C03300=1039.948,345.644,-123.937,172.528,43.194,158.381
C03301=1039.956,345.890,-123.974,172.532,43.197,158.382
C03302=1039.963,346.138,-124.011,172.538,43.201,158.383
C03303=1039.971,346.384,-124.048,172.543,43.204,158.384
C03304=1039.978,346.631,-124.086,172.549,43.206,158.385
C03305=1039.985,346.879,-124.123,172.554,43.209,158.386
C03306=1039.993,347.126,-124.160,172.560,43.213,158.387
C03307=1040.000,347.373,-124.197,172.565,43.215,158.388
C03308=1040.008,347.620,-124.235,172.570,43.218,158.390
C03309=1040.016,347.867,-124.272,172.576,43.221,158.391
C03310=1040.024,348.151,-124.314,172.583,43.225,158.392
C03311=1040.033,348.436,-124.358,172.588,43.228,158.393
C03312=1040.041,348.720,-124.401,172.595,43.232,158.395
C03313=1040.051,349.004,-124.445,172.602,43.236,158.396
C03314=1040.059,349.251,-124.481,172.607,43.238,158.397
C03315=1040.066,349.498,-124.519,172.612,43.242,158.398
C03316=1040.073,349.746,-124.557,172.618,43.245,158.400
C03317=1040.081,349.993,-124.594,172.623,43.248,158.401
C03318=1040.089,350.239,-124.631,172.629,43.251,158.402
C03319=1040.097,350.487,-124.670,172.634,43.254,158.403
C03320=1040.104,350.734,-124.707,172.640,43.257,158.404
C03321=1040.111,350.981,-124.745,172.645,43.261,158.405
C03322=1040.118,351.228,-124.782,172.651,43.263,158.407
C03323=1040.126,351.475,-124.820,172.656,43.267,158.408
C03324=1040.134,351.722,-124.858,172.662,43.270,158.409
C03325=1040.141,351.969,-124.897,172.667,43.273,158.410
C03326=1040.149,352.216,-124.934,172.673,43.276,158.411
C03327=1040.157,352.463,-124.971,172.678,43.280,158.413
C03328=1040.165,352.710,-125.010,172.685,43.282,158.414
C03329=1040.172,352.957,-125.047,172.690,43.286,158.415
C03330=1040.180,353.204,-125.085,172.696,43.289,158.416
C03331=1040.187,353.451,-125.123,172.701,43.293,158.418
C03332=1040.195,353.698,-125.162,172.707,43.296,158.419
C03333=1040.202,353.945,-125.200,172.712,43.299,158.420
C03334=1040.210,354.192,-125.237,172.718,43.302,158.421
C03335=1040.218,354.439,-125.276,172.724,43.306,158.422
C03336=1040.226,354.686,-125.313,172.730,43.309,158.424
C03337=1040.234,354.933,-125.351,172.736,43.312,158.425
C03338=1040.242,355.180,-125.390,172.741,43.316,158.426
C03339=1040.249,355.427,-125.427,172.747,43.319,158.427
C03340=1040.257,355.674,-125.466,172.752,43.322,158.429
C03341=1040.264,355.920,-125.504,172.759,43.325,158.430
C03342=1040.273,356.168,-125.543,172.764,43.329,158.431
C03343=1040.280,356.415,-125.580,172.770,43.332,158.432
C03344=1040.288,356.662,-125.619,172.776,43.335,158.434
C03345=1040.296,356.909,-125.657,172.781,43.339,158.435
C03346=1040.303,357.155,-125.695,172.788,43.342,158.436
C03347=1040.311,357.402,-125.734,172.793,43.345,158.438
C03348=1040.318,357.649,-125.773,172.799,43.349,158.439
C03349=1040.326,357.896,-125.811,172.805,43.353,158.440
C03350=1040.334,358.143,-125.850,172.810,43.356,158.442
C03351=1040.342,358.390,-125.888,172.817,43.359,158.443
C03352=1040.349,358.637,-125.926,172.823,43.363,158.444
C03353=1040.358,358.884,-125.965,172.828,43.366,158.445
C03354=1040.365,359.130,-126.003,172.834,43.370,158.447
C03355=1040.373,359.377,-126.042,172.841,43.373,158.448
C03356=1040.382,359.625,-126.081,172.846,43.377,158.449
C03357=1040.389,359.871,-126.120,172.852,43.381,158.451
C03358=1040.397,360.118,-126.159,172.859,43.384,158.452
C03359=1040.404,360.365,-126.197,172.864,43.387,158.453
C03360=1040.412,360.612,-126.236,172.870,43.391,158.455
C03361=1040.421,360.859,-126.274,172.877,43.394,158.456
C03362=1040.428,361.105,-126.314,172.882,43.398,158.457
C03363=1040.436,361.352,-126.352,172.888,43.402,158.459
C03364=1040.444,361.600,-126.391,172.895,43.405,158.460
C03365=1040.452,361.846,-126.430,172.901,43.409,158.462
C03366=1040.460,362.109,-126.472,172.908,43.413,158.463
C03367=1040.471,362.465,-126.527,172.916,43.418,158.465
C03368=1040.483,362.821,-126.584,172.925,43.423,158.467
C03369=1040.494,363.177,-126.641,172.933,43.429,158.469
C03370=1040.506,363.533,-126.697,172.943,43.434,158.471
C03371=1040.513,363.780,-126.736,172.948,43.437,158.472
C03372=1040.521,364.027,-126.776,172.954,43.441,158.474
C03373=1040.529,364.273,-126.815,172.961,43.445,158.475
C03374=1040.537,364.520,-126.854,172.967,43.449,158.477
C03375=1040.544,364.767,-126.894,172.973,43.452,158.478
C03376=1040.553,365.014,-126.933,172.979,43.456,158.479
C03377=1040.560,365.260,-126.973,172.985,43.460,158.481
C03378=1040.568,365.507,-127.011,172.992,43.464,158.482
C03379=1040.577,365.754,-127.051,172.998,43.468,158.484
C03380=1040.584,366.001,-127.090,173.004,43.471,158.485
C03381=1040.593,366.247,-127.130,173.010,43.475,158.486
C03382=1040.601,366.494,-127.170,173.017,43.479,158.488
C03383=1040.609,366.741,-127.209,173.023,43.482,158.489
C03384=1040.616,366.987,-127.249,173.030,43.486,158.491
C03385=1040.625,367.234,-127.288,173.036,43.490,158.492
C03386=1040.632,367.481,-127.328,173.042,43.494,158.494
C03387=1040.641,367.727,-127.367,173.048,43.498,158.495
C03388=1040.648,367.974,-127.407,173.055,43.502,158.497
C03389=1040.657,368.221,-127.446,173.061,43.505,158.498
C03390=1040.665,368.468,-127.486,173.068,43.509,158.500
C03391=1040.673,368.714,-127.526,173.074,43.513,158.501
C03392=1040.681,368.961,-127.566,173.081,43.517,158.503
C03393=1040.689,369.208,-127.605,173.087,43.521,158.504
C03394=1040.697,369.455,-127.645,173.094,43.525,158.506
C03395=1040.706,369.700,-127.685,173.100,43.529,158.507
C03396=1040.713,369.947,-127.725,173.106,43.533,158.508
C03397=1040.722,370.194,-127.764,173.113,43.537,158.510
C03398=1040.730,370.441,-127.804,173.119,43.541,158.512
C03399=1040.739,370.688,-127.844,173.126,43.545,158.513
C03400=1040.747,370.934,-127.884,173.133,43.549,158.515
C03401=1040.755,371.181,-127.925,173.139,43.553,158.516
C03402=1040.762,371.428,-127.965,173.146,43.557,158.518
C03403=1040.770,371.674,-128.006,173.152,43.561,158.519
C03404=1040.778,371.921,-128.045,173.159,43.565,158.521
C03405=1040.787,372.167,-128.085,173.166,43.569,158.522
C03406=1040.795,372.414,-128.125,173.172,43.574,158.524
C03407=1040.803,372.660,-128.166,173.179,43.577,158.525
C03408=1040.811,372.906,-128.207,173.186,43.582,158.527
C03409=1040.819,373.154,-128.247,173.192,43.586,158.529
C03410=1040.827,373.400,-128.288,173.199,43.590,158.530
C03411=1040.836,373.646,-128.328,173.206,43.594,158.532
C03412=1040.844,373.893,-128.368,173.212,43.598,158.533
C03413=1040.852,374.139,-128.408,173.219,43.602,158.535
C03414=1040.860,374.386,-128.449,173.226,43.607,158.537
C03415=1040.868,374.633,-128.490,173.232,43.611,158.538
C03416=1040.876,374.879,-128.530,173.239,43.615,158.540
C03417=1040.885,375.126,-128.570,173.246,43.619,158.541
C03418=1040.893,375.373,-128.611,173.253,43.623,158.543
C03419=1040.901,375.619,-128.651,173.260,43.628,158.545
C03420=1040.909,375.865,-128.692,173.267,43.632,158.546
C03421=1040.918,376.112,-128.733,173.274,43.636,158.548
C03422=1040.926,376.358,-128.774,173.281,43.640,158.549
C03423=1040.939,376.734,-128.836,173.291,43.647,158.552
C03424=1040.952,377.110,-128.898,173.301,43.654,158.554
C03425=1040.965,377.486,-128.960,173.313,43.660,158.557
C03426=1040.978,377.862,-129.022,173.323,43.667,158.559
C03427=1040.987,378.108,-129.063,173.330,43.671,158.561
C03428=1040.995,378.354,-129.104,173.337,43.676,158.563
C03429=1041.003,378.601,-129.145,173.344,43.680,158.565
C03430=1041.011,378.848,-129.186,173.350,43.684,158.566
C03431=1041.020,379.094,-129.227,173.357,43.689,158.568
C03432=1041.028,379.340,-129.268,173.365,43.693,158.570
C03433=1041.037,379.587,-129.310,173.372,43.698,158.571
C03434=1041.045,379.833,-129.351,173.379,43.702,158.573
C03435=1041.054,380.080,-129.393,173.386,43.707,158.575
C03436=1041.062,380.326,-129.433,173.394,43.711,158.576
C03437=1041.070,380.572,-129.475,173.401,43.716,158.578
C03438=1041.078,380.819,-129.516,173.408,43.720,158.580
C03439=1041.087,381.065,-129.558,173.414,43.725,158.582
C03440=1041.096,381.312,-129.600,173.422,43.729,158.583
C03441=1041.104,381.558,-129.640,173.429,43.734,158.585
C03442=1041.113,381.804,-129.682,173.436,43.738,158.587
C03443=1041.120,382.050,-129.724,173.443,43.743,158.589
C03444=1041.129,382.297,-129.765,173.451,43.748,158.591
C03445=1041.138,382.544,-129.807,173.458,43.752,158.592
C03446=1041.146,382.789,-129.848,173.465,43.757,158.594
C03447=1041.154,383.036,-129.890,173.473,43.762,158.596
C03448=1041.163,383.282,-129.932,173.480,43.767,158.598
C03449=1041.172,383.529,-129.974,173.487,43.771,158.599
C03450=1041.180,383.774,-130.015,173.495,43.776,158.601
C03451=1041.189,384.021,-130.057,173.502,43.781,158.603
C03452=1041.198,384.267,-130.099,173.509,43.785,158.605
C03453=1041.207,384.514,-130.141,173.517,43.790,158.607
C03454=1041.215,384.759,-130.182,173.525,43.795,158.609
C03455=1041.224,385.006,-130.224,173.533,43.800,158.610
C03456=1041.232,385.252,-130.266,173.540,43.804,158.612
C03457=1041.241,385.499,-130.308,173.547,43.809,158.614
C03458=1041.250,385.745,-130.350,173.555,43.814,158.616
C03459=1041.259,385.992,-130.391,173.562,43.819,158.618
C03460=1041.267,386.238,-130.434,173.570,43.823,158.620
C03461=1041.276,386.484,-130.476,173.577,43.828,158.622
C03462=1041.285,386.730,-130.518,173.585,43.833,158.623
C03463=1041.294,386.976,-130.559,173.593,43.838,158.625
C03464=1041.302,387.222,-130.602,173.600,43.842,158.627
C03465=1041.311,387.468,-130.644,173.608,43.848,158.629
C03466=1041.320,387.715,-130.686,173.615,43.852,158.631
C03467=1041.329,387.960,-130.728,173.624,43.857,158.633
C03468=1041.338,388.208,-130.771,173.631,43.862,158.635
C03469=1041.347,388.454,-130.813,173.639,43.867,158.637
C03470=1041.355,388.700,-130.856,173.646,43.872,158.639
C03471=1041.365,388.946,-130.898,173.654,43.877,158.641
C03472=1041.373,389.192,-130.941,173.662,43.882,158.642
C03473=1041.382,389.438,-130.983,173.670,43.887,158.644
C03474=1041.391,389.684,-131.026,173.677,43.892,158.646
C03475=1041.400,389.930,-131.068,173.686,43.897,158.648
C03476=1041.408,390.176,-131.111,173.694,43.902,158.650
C03477=1041.417,390.423,-131.153,173.701,43.908,158.652
C03478=1041.426,390.669,-131.196,173.709,43.912,158.654
C03479=1041.440,391.079,-131.267,173.722,43.921,158.658
C03480=1041.456,391.489,-131.339,173.735,43.930,158.661
C03481=1041.470,391.898,-131.410,173.749,43.938,158.664
C03482=1041.485,392.308,-131.482,173.762,43.947,158.668
C03483=1041.495,392.554,-131.525,173.770,43.952,158.670
C03484=1041.503,392.801,-131.568,173.779,43.958,158.672
C03485=1041.512,393.047,-131.611,173.786,43.963,158.674
C03486=1041.521,393.292,-131.654,173.795,43.968,158.676
C03487=1041.530,393.538,-131.697,173.803,43.973,158.678
C03488=1041.539,393.785,-131.740,173.811,43.978,158.680
C03489=1041.547,394.031,-131.783,173.819,43.984,158.682
C03490=1041.557,394.276,-131.827,173.827,43.989,158.684
C03491=1041.566,394.522,-131.870,173.836,43.995,158.686
C03492=1041.574,394.769,-131.913,173.843,44.000,158.688
C03493=1041.585,395.014,-131.956,173.852,44.005,158.690
C03494=1041.593,395.260,-131.999,173.860,44.011,158.693
C03495=1041.602,395.507,-132.044,173.869,44.016,158.695
C03496=1041.611,395.753,-132.087,173.877,44.022,158.697
C03497=1041.620,395.999,-132.131,173.885,44.027,158.699
C03498=1041.630,396.244,-132.174,173.894,44.032,158.701
C03499=1041.639,396.491,-132.217,173.902,44.038,158.703
C03500=1041.648,396.736,-132.261,173.911,44.043,158.705
C03501=1041.657,396.982,-132.305,173.919,44.049,158.708
C03502=1041.666,397.228,-132.349,173.927,44.054,158.710
C03503=1041.675,397.474,-132.392,173.936,44.060,158.712
C03504=1041.684,397.720,-132.436,173.944,44.066,158.714
C03505=1041.693,397.966,-132.480,173.953,44.071,158.716
C03506=1041.702,398.211,-132.524,173.961,44.077,158.718
C03507=1041.712,398.457,-132.567,173.970,44.082,158.721
C03508=1041.722,398.703,-132.611,173.979,44.088,158.723
C03509=1041.731,398.949,-132.655,173.987,44.094,158.725
C03510=1041.740,399.195,-132.699,173.996,44.099,158.727
C03511=1041.749,399.441,-132.743,174.005,44.105,158.730
C03512=1041.759,399.687,-132.787,174.014,44.110,158.732
C03513=1041.768,399.933,-132.831,174.022,44.116,158.734
C03514=1041.777,400.179,-132.875,174.031,44.122,158.736
C03515=1041.787,400.424,-132.920,174.040,44.128,158.739
C03516=1041.796,400.670,-132.964,174.049,44.134,158.741
C03517=1041.805,400.916,-133.008,174.057,44.139,158.743
C03518=1041.815,401.161,-133.053,174.066,44.145,158.746
C03519=1041.824,401.407,-133.097,174.075,44.151,158.748
C03520=1041.833,401.654,-133.141,174.084,44.157,158.750
C03521=1041.842,401.899,-133.186,174.092,44.163,158.753
C03522=1041.852,402.146,-133.231,174.101,44.169,158.755
C03523=1041.862,402.391,-133.275,174.110,44.175,158.757
C03524=1041.871,402.637,-133.319,174.119,44.180,158.760
C03525=1041.881,402.883,-133.364,174.128,44.186,158.762
C03526=1041.890,403.128,-133.409,174.137,44.192,158.764
C03527=1041.899,403.375,-133.454,174.147,44.198,158.767
C03528=1041.909,403.620,-133.499,174.156,44.204,158.769
C03529=1041.918,403.866,-133.543,174.164,44.211,158.772
C03530=1041.928,404.111,-133.588,174.173,44.216,158.774
C03531=1041.937,404.358,-133.633,174.182,44.222,158.776
C03532=1041.947,404.603,-133.678,174.192,44.228,158.779
C03533=1041.956,404.849,-133.723,174.201,44.235,158.781
C03534=1041.965,405.094,-133.768,174.210,44.241,158.784
C03535=1041.974,405.309,-133.807,174.218,44.246,158.786
C03536=1041.982,405.524,-133.847,174.227,44.251,158.788
C03537=1041.991,405.739,-133.886,174.235,44.257,158.790
C03538=1041.999,405.953,-133.925,174.243,44.262,158.792
C03539=1042.007,406.168,-133.965,174.250,44.267,158.794
C03540=1042.016,406.382,-134.005,174.259,44.273,158.797
C03541=1042.024,406.597,-134.044,174.267,44.279,158.799
C03542=1042.032,406.812,-134.084,174.275,44.284,158.801
C03543=1042.042,407.058,-134.129,174.285,44.291,158.803
C03544=1042.052,407.303,-134.175,174.295,44.296,158.806
C03545=1042.061,407.549,-134.220,174.304,44.302,158.808
C03546=1042.071,407.795,-134.265,174.314,44.309,158.811
C03547=1042.081,408.040,-134.312,174.323,44.315,158.813
C03548=1042.090,408.286,-134.356,174.333,44.322,158.816
C03549=1042.101,408.532,-134.402,174.342,44.328,158.819
C03550=1042.110,408.777,-134.448,174.352,44.334,158.821
C03551=1042.120,409.023,-134.493,174.362,44.341,158.824
C03552=1042.130,409.268,-134.539,174.371,44.347,158.826
C03553=1042.140,409.513,-134.585,174.381,44.354,158.829
C03554=1042.150,409.760,-134.630,174.391,44.360,158.832
C03555=1042.159,410.005,-134.676,174.401,44.367,158.834
C03556=1042.170,410.250,-134.722,174.410,44.373,158.837
C03557=1042.179,410.497,-134.768,174.420,44.380,158.840
C03558=1042.190,410.742,-134.813,174.430,44.386,158.842
C03559=1042.200,410.987,-134.859,174.440,44.392,158.845
C03560=1042.209,411.233,-134.905,174.450,44.399,158.848
C03561=1042.220,411.478,-134.951,174.460,44.406,158.850
C03562=1042.230,411.724,-134.998,174.470,44.412,158.853
C03563=1042.241,411.970,-135.043,174.480,44.419,158.855
C03564=1042.250,412.215,-135.090,174.490,44.425,158.858
C03565=1042.260,412.461,-135.136,174.501,44.432,158.861
C03566=1042.270,412.706,-135.182,174.510,44.439,158.864
C03567=1042.280,412.952,-135.228,174.520,44.446,158.866
C03568=1042.290,413.197,-135.275,174.530,44.452,158.869
C03569=1042.300,413.443,-135.322,174.540,44.459,158.872
C03570=1042.310,413.688,-135.368,174.551,44.466,158.875
C03571=1042.320,413.933,-135.415,174.561,44.473,158.877
C03572=1042.330,414.179,-135.461,174.572,44.480,158.880
C03573=1042.340,414.425,-135.508,174.582,44.486,158.883
C03574=1042.351,414.670,-135.554,174.592,44.493,158.886
C03575=1042.361,414.916,-135.601,174.603,44.500,158.889
C03576=1042.371,415.161,-135.648,174.613,44.507,158.892
C03577=1042.381,415.406,-135.695,174.623,44.514,158.894
C03578=1042.392,415.652,-135.741,174.634,44.521,158.897
C03579=1042.402,415.897,-135.788,174.644,44.528,158.900
C03580=1042.412,416.142,-135.836,174.655,44.535,158.903
C03581=1042.422,416.388,-135.883,174.666,44.542,158.906
C03582=1042.432,416.634,-135.929,174.676,44.549,158.909
C03583=1042.443,416.878,-135.976,174.687,44.556,158.912
C03584=1042.453,417.124,-136.023,174.698,44.563,158.915
C03585=1042.463,417.369,-136.070,174.709,44.570,158.917
C03586=1042.473,417.614,-136.118,174.719,44.578,158.921
C03587=1042.484,417.860,-136.165,174.730,44.584,158.923
C03588=1042.495,418.105,-136.212,174.741,44.592,158.926
C03589=1042.505,418.351,-136.259,174.752,44.599,158.929
C03590=1042.516,418.596,-136.306,174.763,44.606,158.932
C03591=1042.526,418.841,-136.354,174.774,44.613,158.935
C03592=1042.536,419.086,-136.401,174.784,44.620,158.938
C03593=1042.547,419.332,-136.449,174.795,44.628,158.941
C03594=1042.557,419.577,-136.497,174.806,44.635,158.944
C03595=1042.567,419.795,-136.540,174.817,44.641,158.947
C03596=1042.576,420.014,-136.582,174.827,44.648,158.950
C03597=1042.585,420.233,-136.625,174.836,44.655,158.953
C03598=1042.595,420.452,-136.667,174.846,44.661,158.955
C03599=1042.604,420.671,-136.710,174.856,44.668,158.958
C03600=1042.614,420.890,-136.752,174.866,44.674,158.961
C03601=1042.622,421.107,-136.795,174.876,44.681,158.964
C03602=1042.632,421.326,-136.838,174.886,44.688,158.967
C03603=1042.643,421.571,-136.886,174.897,44.695,158.970
C03604=1042.654,421.816,-136.934,174.910,44.703,158.973
C03605=1042.664,422.062,-136.982,174.921,44.710,158.976
C03606=1042.674,422.307,-137.030,174.932,44.718,158.979
C03607=1042.685,422.552,-137.078,174.943,44.725,158.982
C03608=1042.697,422.798,-137.127,174.955,44.733,158.986
C03609=1042.707,423.042,-137.175,174.966,44.741,158.989
